(* CoDeSys 2.3.9.47 project: samur_8_8_16.pro *)
(* Libraries: STANDARD.LIB 5.6.98 12:03:02 *)

(* Task configuration *)
TASK Standard (PRIORITY := 0, INTERVAL := T#10ms);
	MAIN
END_TASK

(* Global variable list: TwinCAT_Configuration *)
(* Generated automatically by TwinCAT - (read only) *)
VAR_CONFIG
	CCB_FirstFloor.FCU_CCB1_23A_status AT %IX9.4 : BOOL;
	CCB_FirstFloor.FCU_CCB1_23A_trip AT %IX9.5 : BOOL;
	CCB_FirstFloor.FCU_CCB1_23A_mode AT %IX9.6 : BOOL;
	CCB_FirstFloor.FCU_CCB1_23A_FB.DEV1.AHU1_Relay AT %QX3.4 : BOOL;
	CCB_FirstFloor.FCU_CCB1_23B_status AT %IX9.7 : BOOL;
	CCB_FirstFloor.FCU_CCB1_23B_trip AT %IX10.0 : BOOL;
	CCB_FirstFloor.FCU_CCB1_23B_mode AT %IX10.1 : BOOL;
	CCB_FirstFloor.FCU_CCB1_23B_FB.DEV1.AHU1_Relay AT %QX3.5 : BOOL;
	CCB_FirstFloor.FCU_CCB1_23C_status AT %IX10.2 : BOOL;
	CCB_FirstFloor.FCU_CCB1_23C_trip AT %IX10.3 : BOOL;
	CCB_FirstFloor.FCU_CCB1_23C_mode AT %IX10.4 : BOOL;
	CCB_FirstFloor.FCU_CCB1_23C_FB.DEV1.AHU1_Relay AT %QX3.6 : BOOL;
	CCB_FirstFloor.DCS_Occupied AT %QX0.2 : BOOL;
	CCB_FirstFloor.common_alarm AT %QX0.3 : BOOL;
	CCB_GroundFloor.AHU_CCBG_01_status AT %IX0.0 : BOOL;
	CCB_GroundFloor.AHU_CCBG_01_trip AT %IX0.1 : BOOL;
	CCB_GroundFloor.AHU_CCBG_01_mode AT %IX0.2 : BOOL;
	CCB_GroundFloor.AHU_CCBG_01_belt AT %IX0.3 : BOOL;
	CCB_GroundFloor.AHU_CCBG_01_fire AT %IX0.4 : BOOL;
	CCB_GroundFloor.AHU_CCBG_01_gas AT %IX0.5 : BOOL;
	CCB_GroundFloor.AHU_CCBG_01_smoke AT %IX0.6 : BOOL;
	CCB_GroundFloor.AHU_CCBG_02_status AT %IX0.7 : BOOL;
	CCB_GroundFloor.AHU_CCBG_02_trip AT %IX1.0 : BOOL;
	CCB_GroundFloor.AHU_CCBG_02_mode AT %IX1.1 : BOOL;
	CCB_GroundFloor.AHU_CCBG_02_belt AT %IX1.2 : BOOL;
	CCB_GroundFloor.AHU_CCBG_02_fire AT %IX1.3 : BOOL;
	CCB_GroundFloor.AHU_CCBG_02_gas AT %IX1.4 : BOOL;
	CCB_GroundFloor.AHU_CCBG_02_smoke AT %IX1.5 : BOOL;
	CCB_GroundFloor.AHU_CCBG_03_status AT %IX1.6 : BOOL;
	CCB_GroundFloor.AHU_CCBG_03_trip AT %IX1.7 : BOOL;
	CCB_GroundFloor.AHU_CCBG_03_mode AT %IX2.0 : BOOL;
	CCB_GroundFloor.AHU_CCBG_03_belt AT %IX2.1 : BOOL;
	CCB_GroundFloor.AHU_CCBG_03_fire AT %IX2.2 : BOOL;
	CCB_GroundFloor.AHU_CCBG_03_gas AT %IX2.3 : BOOL;
	CCB_GroundFloor.AHU_CCBG_03_smoke AT %IX2.4 : BOOL;
	CCB_GroundFloor.AHU_CCCBG.DEV_1.AHU1_Relay AT %QX1.7 : BOOL;
	CCB_GroundFloor.AHU_CCCBG.DEV_2.AHU1_Relay AT %QX2.0 : BOOL;
	CCB_GroundFloor.AHU_CCCBG.DEV_3.AHU1_Relay AT %QX2.1 : BOOL;
	CCB_GroundFloor.EF_CCB_1_status AT %IX2.5 : BOOL;
	CCB_GroundFloor.EF_CCB_1_trip AT %IX2.6 : BOOL;
	CCB_GroundFloor.EF_CCB_1_mode AT %IX2.7 : BOOL;
	CCB_GroundFloor.EF_CCB_2_status AT %IX3.0 : BOOL;
	CCB_GroundFloor.EF_CCB_2_trip AT %IX3.1 : BOOL;
	CCB_GroundFloor.EF_CCB_2_mode AT %IX3.2 : BOOL;
	CCB_GroundFloor.EF_CCB.DEV_1.AHU1_Relay AT %QX2.2 : BOOL;
	CCB_GroundFloor.EF_CCB.DEV_2.AHU1_Relay AT %QX2.3 : BOOL;
	CCB_GroundFloor.TEF_CCB_01_status AT %IX3.3 : BOOL;
	CCB_GroundFloor.TEF_CCB_01_trip AT %IX3.4 : BOOL;
	CCB_GroundFloor.TEF_CCB_01_mode AT %IX3.5 : BOOL;
	CCB_GroundFloor.TEC_CCB.DEV1.AHU1_Relay AT %QX2.5 : BOOL;
	CCB_GroundFloor.EF_CCB_7A_status AT %IX3.6 : BOOL;
	CCB_GroundFloor.EF_CCB_7A_trip AT %IX3.7 : BOOL;
	CCB_GroundFloor.EF_CCB_7B_status AT %IX4.0 : BOOL;
	CCB_GroundFloor.EF_CCB_7B_trip AT %IX4.1 : BOOL;
	CCB_GroundFloor.EF_CCB_08_status AT %IX4.2 : BOOL;
	CCB_GroundFloor.EF_CCB_08_trip AT %IX4.3 : BOOL;
	CCB_GroundFloor.EH_CCB_01_flow_status AT %IX4.5 : BOOL;
	CCB_GroundFloor.EH_CCB_01_high_temp AT %IX4.6 : BOOL;
	CCB_GroundFloor.EH_CCB_01_FB.TEMPERATURE AT %IB32 : INT;
	CCB_GroundFloor.EH_CCB_01_FB.HEATER_STAGE1 AT %QX2.6 : BOOL;
	CCB_GroundFloor.EH_CCB_01_FB.HEATER_STAGE2 AT %QX2.7 : BOOL;
	CCB_GroundFloor.EH_CCB_01_FB.HEATER_STAGE3 AT %QX3.0 : BOOL;
	CCB_GroundFloor.EH_CCB_02_flow_status AT %IX5.0 : BOOL;
	CCB_GroundFloor.EH_CCB_02_high_temp AT %IX5.1 : BOOL;
	CCB_GroundFloor.EH_CCB_02_FB.TEMPERATURE AT %IB34 : INT;
	CCB_GroundFloor.EH_CCB_02_FB.HEATER_STAGE1 AT %QX3.1 : BOOL;
	CCB_GroundFloor.EH_CCB_02_FB.HEATER_STAGE2 AT %QX3.2 : BOOL;
	CCB_GroundFloor.EH_CCB_02_FB.HEATER_STAGE3 AT %QX3.3 : BOOL;
	CCB_GroundFloor.MD_CCBG_1_damper_open AT %IX5.2 : BOOL;
	CCB_GroundFloor.MD_CCBG_1_damper_close AT %IX5.3 : BOOL;
	CCB_GroundFloor.MD_CCBG_2_damper_open AT %IX5.4 : BOOL;
	CCB_GroundFloor.MD_CCBG_2_damper_close AT %IX5.5 : BOOL;
	CCB_GroundFloor.MD_CCBG_3_damper_open AT %IX5.6 : BOOL;
	CCB_GroundFloor.MD_CCBG_3_damper_close AT %IX5.7 : BOOL;
	CCB_GroundFloor.MD_CCBG_4_damper_open AT %IX6.0 : BOOL;
	CCB_GroundFloor.MD_CCBG_4_damper_close AT %IX6.1 : BOOL;
	CCB_GroundFloor.MD_EF_CCB_7A_damper_open AT %IX6.2 : BOOL;
	CCB_GroundFloor.MD_EF_CCB_7A_damper_close AT %IX6.3 : BOOL;
	CCB_GroundFloor.MD_EF_CCB_7B_damper_open AT %IX6.4 : BOOL;
	CCB_GroundFloor.MD_EF_CCB_7B_damper_close AT %IX6.5 : BOOL;
	CCB_GroundFloor.MD_EF_CCB_8_damper_open AT %IX6.6 : BOOL;
	CCB_GroundFloor.MD_EF_CCB_8_damper_close AT %IX6.7 : BOOL;
	CCB_GroundFloor.MFD_CCB_1_damper_open AT %IX7.0 : BOOL;
	CCB_GroundFloor.MFD_CCB_1_damper_close AT %IX7.1 : BOOL;
	CCB_GroundFloor.MFD_CCB_2_damper_open AT %IX7.2 : BOOL;
	CCB_GroundFloor.MFD_CCB_2_damper_close AT %IX7.3 : BOOL;
	CCB_GroundFloor.MFD_CCB_3_damper_open AT %IX7.4 : BOOL;
	CCB_GroundFloor.MFD_CCB_3_damper_close AT %IX7.5 : BOOL;
	CCB_GroundFloor.MFD_CCB_4_damper_open AT %IX7.6 : BOOL;
	CCB_GroundFloor.MFD_CCB_4_damper_close AT %IX7.7 : BOOL;
	CCB_GroundFloor.MFD_CCB_5_damper_open AT %IX8.0 : BOOL;
	CCB_GroundFloor.MFD_CCB_5_damper_close AT %IX8.1 : BOOL;
	CCB_GroundFloor.MFD_CCB_6_damper_open AT %IX8.2 : BOOL;
	CCB_GroundFloor.MFD_CCB_6_damper_close AT %IX8.3 : BOOL;
	CCB_GroundFloor.MFD_CCB_7_damper_open AT %IX8.4 : BOOL;
	CCB_GroundFloor.MFD_CCB_7_damper_close AT %IX8.5 : BOOL;
	CCB_GroundFloor.MFD_CCB_8_damper_open AT %IX8.6 : BOOL;
	CCB_GroundFloor.MFD_CCB_8_damper_close AT %IX8.7 : BOOL;
	CCB_GroundFloor.MFD_CCB_9_damper_open AT %IX9.0 : BOOL;
	CCB_GroundFloor.MFD_CCB_9_damper_close AT %IX9.1 : BOOL;
	CCB_GroundFloor.MFD_CCB_10_damper_open AT %IX9.2 : BOOL;
	CCB_GroundFloor.MFD_CCB_10_damper_close AT %IX9.3 : BOOL;
	CCB_GroundFloor.DCS_Occupied AT %QX0.0 : BOOL;
	CCB_GroundFloor.common_alarm AT %QX0.1 : BOOL;
	EDG_HOUSE.FB_AHU_EDG.DEV_1.AHU1_Relay AT %QX3.7 : BOOL;
	EDG_HOUSE.FB_AHU_EDG.DEV_2.AHU1_Relay AT %QX4.0 : BOOL;
	EDG_HOUSE.AHU_EDG_1_status AT %IX24.0 : BOOL;
	EDG_HOUSE.AHU_EDG_1_trip AT %IX24.1 : BOOL;
	EDG_HOUSE.AHU_EDG_1_mode AT %IX24.2 : BOOL;
	EDG_HOUSE.AHU_EDG_1_belt AT %IX24.3 : BOOL;
	EDG_HOUSE.AHU_EDG_1_fire AT %IX24.4 : BOOL;
	EDG_HOUSE.AHU_EDG_1_gas AT %IX24.5 : BOOL;
	EDG_HOUSE.AHU_EDG_1_smoke AT %IX24.6 : BOOL;
	EDG_HOUSE.AHU_EDG_2_status AT %IX24.7 : BOOL;
	EDG_HOUSE.AHU_EDG_2_trip AT %IX25.0 : BOOL;
	EDG_HOUSE.AHU_EDG_2_mode AT %IX25.1 : BOOL;
	EDG_HOUSE.AHU_EDG_2_belt AT %IX25.2 : BOOL;
	EDG_HOUSE.AHU_EDG_2_fire AT %IX25.3 : BOOL;
	EDG_HOUSE.AHU_EDG_2_gas AT %IX25.4 : BOOL;
	EDG_HOUSE.AHU_EDG_2_smoke AT %IX25.5 : BOOL;
	EDG_HOUSE.FB_EF_EDG.DEV_1.AHU1_Relay AT %QX4.2 : BOOL;
	EDG_HOUSE.FB_EF_EDG.DEV_2.AHU1_Relay AT %QX4.3 : BOOL;
	EDG_HOUSE.EF_EDG_1A_status AT %IX26.5 : BOOL;
	EDG_HOUSE.EF_EDG_1A_trip AT %IX26.6 : BOOL;
	EDG_HOUSE.EF_EDG_1A_mode AT %IX26.7 : BOOL;
	EDG_HOUSE.EF_EDG_1B_status AT %IX27.0 : BOOL;
	EDG_HOUSE.EF_EDG_1B_trip AT %IX27.1 : BOOL;
	EDG_HOUSE.EF_EDG_1B_mode AT %IX27.2 : BOOL;
	EDG_HOUSE.EF_EDG_2_status AT %IX27.3 : BOOL;
	EDG_HOUSE.EF_EDG_2_trip AT %IX27.4 : BOOL;
	EDG_HOUSE.EF_EDG_2_mode AT %IX27.5 : BOOL;
	EDG_HOUSE.MD_EDG_1A_damper_open AT %IX27.6 : BOOL;
	EDG_HOUSE.MD_EDG_1A_damper_close AT %IX27.7 : BOOL;
	EDG_HOUSE.MD_EDG_1B_damper_open AT %IX28.0 : BOOL;
	EDG_HOUSE.MD_EDG_1B_damper_close AT %IX28.1 : BOOL;
	EDG_HOUSE.MD_EF_EDG_2_damper_open AT %IX28.2 : BOOL;
	EDG_HOUSE.MD_EF_EDG_2_damper_close AT %IX28.3 : BOOL;
	EDG_HOUSE.MFD_EDG_1_damper_open AT %IX28.4 : BOOL;
	EDG_HOUSE.MFD_EDG_1_damper_close AT %IX28.5 : BOOL;
	EDG_HOUSE.MFD_EDG_2_damper_open AT %IX28.6 : BOOL;
	EDG_HOUSE.MFD_EDG_2_damper_close AT %IX28.7 : BOOL;
	EDG_HOUSE.MFD_EDG_3_damper_open AT %IX29.0 : BOOL;
	EDG_HOUSE.MFD_EDG_3_damper_close AT %IX29.1 : BOOL;
	Laboratory.AHU_LAB_1_status AT %IX10.5 : BOOL;
	Laboratory.AHU_LAB_1_trip AT %IX10.6 : BOOL;
	Laboratory.AHU_LAB_1_mode AT %IX10.7 : BOOL;
	Laboratory.AHU_LAB_1_belt AT %IX11.0 : BOOL;
	Laboratory.AHU_LAB_1_fire AT %IX11.1 : BOOL;
	Laboratory.AHU_LAB_1_gas AT %IX11.2 : BOOL;
	Laboratory.AHU_LAB_1_smoke AT %IX11.3 : BOOL;
	Laboratory.AHU_LAB_2_status AT %IX11.4 : BOOL;
	Laboratory.AHU_LAB_2_trip AT %IX11.5 : BOOL;
	Laboratory.AHU_LAB_2_mode AT %IX11.6 : BOOL;
	Laboratory.AHU_LAB_2_belt AT %IX11.7 : BOOL;
	Laboratory.AHU_LAB_2_fire AT %IX12.0 : BOOL;
	Laboratory.AHU_LAB_2_gas AT %IX12.1 : BOOL;
	Laboratory.AHU_LAB_2_smoke AT %IX12.2 : BOOL;
	Laboratory.AHU_LAB_3_status AT %IX12.3 : BOOL;
	Laboratory.AHU_LAB_3_trip AT %IX12.4 : BOOL;
	Laboratory.AHU_LAB_3_mode AT %IX12.5 : BOOL;
	Laboratory.AHU_LAB_3_belt AT %IX12.6 : BOOL;
	Laboratory.AHU_LAB_3_fire AT %IX12.7 : BOOL;
	Laboratory.AHU_LAB_3_gas AT %IX13.0 : BOOL;
	Laboratory.AHU_LAB_3_smoke AT %IX13.1 : BOOL;
	Laboratory.EF_LAB_1_status AT %IX13.2 : BOOL;
	Laboratory.EF_LAB_1_trip AT %IX13.3 : BOOL;
	Laboratory.EF_LAB_1_mode AT %IX13.4 : BOOL;
	Laboratory.EF_LAB_2_status AT %IX13.5 : BOOL;
	Laboratory.EF_LAB_2_trip AT %IX13.6 : BOOL;
	Laboratory.EF_LAB_2_mode AT %IX13.7 : BOOL;
	Laboratory.EF_LAB_3_status AT %IX14.0 : BOOL;
	Laboratory.EF_LAB_3_trip AT %IX14.1 : BOOL;
	Laboratory.EF_LAB_3_mode AT %IX14.2 : BOOL;
	Laboratory.EH_LAB_1_flow_status AT %IX14.4 : BOOL;
	Laboratory.EH_LAB_1_high_temp AT %IX14.5 : BOOL;
	Laboratory.MD_LAB_1_damper_open AT %IX14.6 : BOOL;
	Laboratory.MD_LAB_1_damper_close AT %IX14.7 : BOOL;
	Laboratory.MD_LAB_2_damper_open AT %IX15.0 : BOOL;
	Laboratory.MD_LAB_2_damper_close AT %IX15.1 : BOOL;
	Laboratory.MD_LAB_3_damper_open AT %IX15.2 : BOOL;
	Laboratory.MD_LAB_3_damper_close AT %IX15.3 : BOOL;
	Laboratory.MD_LAB_4_damper_open AT %IX15.4 : BOOL;
	Laboratory.MD_LAB_4_damper_close AT %IX15.5 : BOOL;
	TEST.fbTest_Flowchart_1_2.bAHU1_Status AT %IX29.2 : BOOL;
	TEST.fbTest_Flowchart_1_2.bAHU1_Trip AT %IX29.3 : BOOL;
	TEST.fbTest_Flowchart_1_2.bAHU1_Relay AT %QX0.4 : BOOL;
	TEST.fbTest_Flowchart_1_2.bAHU2_Status AT %IX29.4 : BOOL;
	TEST.fbTest_Flowchart_1_2.bAHU2_Trip AT %IX29.5 : BOOL;
	TEST.fbTest_Flowchart_1_2.bAHU2_Relay AT %QX0.5 : BOOL;
	TEST.fbTest_Flowchart_1_2.AHU1_DcsOccupied AT %QX0.6 : BOOL;
	TEST.fbTest_Flowchart_1_2.AHU1_StatusError AT %QX0.7 : BOOL;
	TEST.fbTest_Flowchart_1_2.AHU1_TripError AT %QX1.0 : BOOL;
	TEST.fbTest_Flowchart_1_2.AHU2_DcsOccupied AT %QX1.1 : BOOL;
	TEST.fbTest_Flowchart_1_2.AHU2_StatusError AT %QX1.2 : BOOL;
	TEST.fbTest_Flowchart_1_2.AHU2_TripError AT %QX1.3 : BOOL;
	TEST.fbtest.TEMPERATURE AT %IB30 : INT;
	TEST.fbtest.HEATER_STAGE1 AT %QX1.4 : BOOL;
	TEST.fbtest.HEATER_STAGE2 AT %QX1.5 : BOOL;
	TEST.fbtest.HEATER_STAGE3 AT %QX1.6 : BOOL;
END_VAR

(* POU MAIN, CFC *)
PROGRAM MAIN
VAR
END_VAR
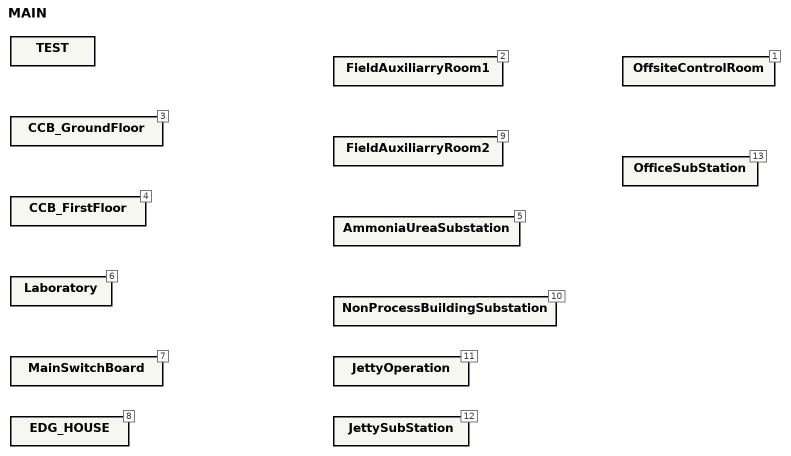
_CFC_ (* Continuous Function Chart, elements in execution order *)
#0 TEST()
#1 OffsiteControlRoom()
#2 FieldAuxiliarryRoom1()
#3 CCB_GroundFloor()
#4 CCB_FirstFloor()
#5 AmmoniaUreaSubstation()
#6 Laboratory()
#7 MainSwitchBoard()
#8 EDG_HOUSE()
#9 FieldAuxiliarryRoom2()
#10 NonProcessBuildingSubstation()
#11 JettyOperation()
#12 JettySubStation()
#13 OfficeSubStation()
_END_CFC_
(* the same logic as Structured Text *)
TEST();
OffsiteControlRoom();
FieldAuxiliarryRoom1();
CCB_GroundFloor();
CCB_FirstFloor();
AmmoniaUreaSubstation();
Laboratory();
MainSwitchBoard();
EDG_HOUSE();
FieldAuxiliarryRoom2();
NonProcessBuildingSubstation();
JettyOperation();
JettySubStation();
OfficeSubStation();
END_PROGRAM

(* POU GarbageCan/TEST, CFC *)
PROGRAM TEST
VAR
	fbTest_Flowchart_1_2: Flowchart_3_4_SingleButton;
	bAHU1: BOOL;
	bAHU2: BOOL;
	bAHU3: BOOL;

	fbtest: Flowchart_5_6;
END_VAR
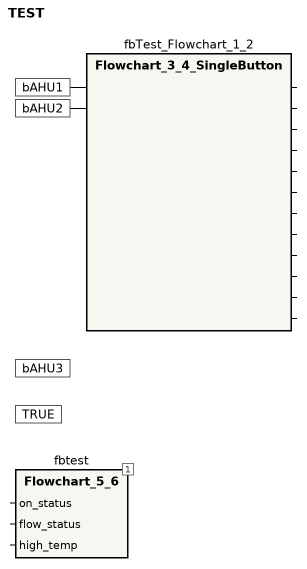
_CFC_ (* Continuous Function Chart, elements in execution order *)
#0 fbTest_Flowchart_1_2:Flowchart_3_4_SingleButton(bAHU1, bAHU2)
unconnected input bAHU3
unconnected input TRUE
#1 fbtest:Flowchart_5_6(on_status: -, flow_status: -, high_temp: -)
_END_CFC_
(* the same logic as Structured Text *)
fbTest_Flowchart_1_2(bAHU1, bAHU2);
fbtest();
END_PROGRAM

(* POU GarbageCan/Flowchart_3_4_SingleButton, CFC *)
FUNCTION_BLOCK Flowchart_3_4_SingleButton
VAR_INPUT
END_VAR
VAR_OUTPUT
	AHU1_DcsOccupied AT%Q*: BOOL;
	AHU1_StatusError  AT%Q*: BOOL;
	AHU1_TripError AT%Q*: BOOL;
	bAHU1_Error: BOOL;

	AHU2_DcsOccupied AT%Q*: BOOL;
	AHU2_StatusError  AT%Q*: BOOL;
	AHU2_TripError AT%Q*: BOOL;
	bAHU2_Error: BOOL;

	AHU_CommonAlarm:BOOL;
	AHU_DCSOccupied:BOOL;

END_VAR
VAR




	bAHU1_Status AT %I*: BOOL;
	bAHU1_Trip AT %I*: BOOL;
	bAHU1_Relay AT %Q*: BOOL;
	Status_timer_1: TON;
	Error_timer_1: TOF;
	OnRtrigAHU1: R_TRIG;
	OffRtrigAHU1: R_TRIG;


	bAHU2_Status AT %I*: BOOL;
	bAHU2_Trip AT %I*: BOOL;
	bAHU2_Relay AT %Q*: BOOL;
	Status_timer_2: TON;
	Error_timer_2: TOF;
	OnRtrigAHU2: R_TRIG;
	OffRtrigAHU2: R_TRIG;


	AHU1_Reset: TON;
	AHU2_Reset: TON;
END_VAR
VAR_IN_OUT
	bAHU1_On: BOOL;
	bAHU2_On: BOOL;

END_VAR
VAR (* helpers for the ST form of the networks *)
	_t14 : BOOL;
	_t65 : BOOL;
	_t137 : BOOL;
	_t152 : BOOL;
END_VAR
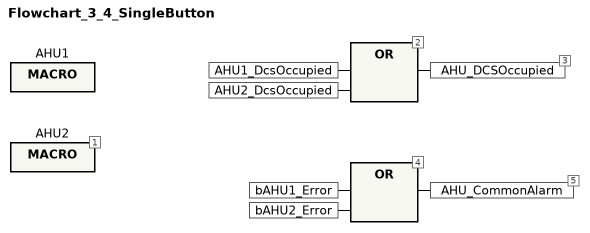
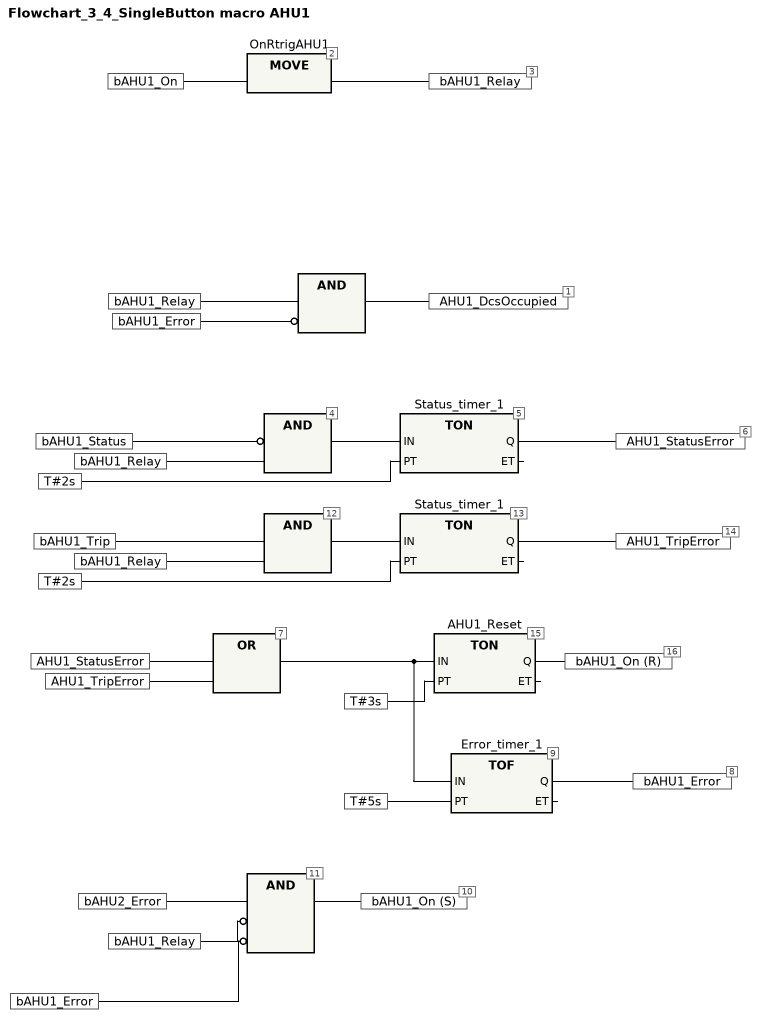
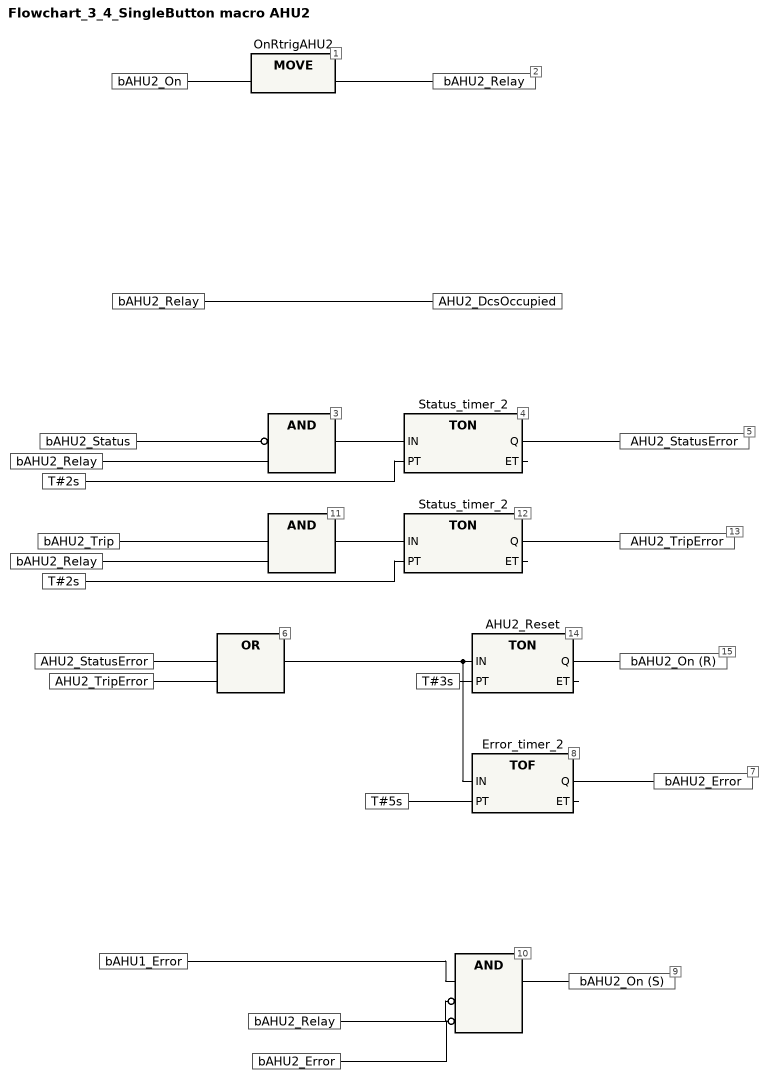
_CFC_ (* Continuous Function Chart, elements in execution order *)
#0 MACRO AHU1()
	#1 AND(bAHU1_Relay, NOT bAHU1_Error)
	#2 AHU1_DcsOccupied <= #1
	#3 OnRtrigAHU1:MOVE(bAHU1_On)
	#4 bAHU1_Relay <= #3
	#5 AND(NOT bAHU1_Status, bAHU1_Relay)
	#6 Status_timer_1:TON(IN: #5, PT: T#2s)
	#7 AHU1_StatusError <= #6.Q
	#8 OR(AHU1_StatusError, AHU1_TripError)
	#9 bAHU1_Error <= #10.Q
	#10 Error_timer_1:TOF(IN: #8, PT: T#5s)
	#11 S bAHU1_On <= #12
	#12 AND(bAHU2_Error, NOT bAHU1_Relay, NOT bAHU1_Error)
	#13 AND(bAHU1_Trip, bAHU1_Relay)
	#14 Status_timer_1:TON(IN: #13, PT: T#2s)
	#15 AHU1_TripError <= #14.Q
	#16 AHU1_Reset:TON(IN: #8, PT: T#3s)
	#17 R bAHU1_On <= #16.Q
END_MACRO
#18 MACRO AHU2()
	#19 AHU2_DcsOccupied <= bAHU2_Relay
	#20 OnRtrigAHU2:MOVE(bAHU2_On)
	#21 bAHU2_Relay <= #20
	#22 AND(NOT bAHU2_Status, bAHU2_Relay)
	#23 Status_timer_2:TON(IN: #22, PT: T#2s)
	#24 AHU2_StatusError <= #23.Q
	#25 OR(AHU2_StatusError, AHU2_TripError)
	#26 bAHU2_Error <= #27.Q
	#27 Error_timer_2:TOF(IN: #25, PT: T#5s)
	#28 S bAHU2_On <= #29
	#29 AND(bAHU1_Error, NOT bAHU2_Relay, NOT bAHU2_Error)
	#30 AND(bAHU2_Trip, bAHU2_Relay)
	#31 Status_timer_2:TON(IN: #30, PT: T#2s)
	#32 AHU2_TripError <= #31.Q
	#33 AHU2_Reset:TON(IN: #25, PT: T#3s)
	#34 R bAHU2_On <= #33.Q
END_MACRO
#35 OR(AHU1_DcsOccupied, AHU2_DcsOccupied)
#36 AHU_DCSOccupied <= #35
#37 OR(bAHU1_Error, bAHU2_Error)
#38 AHU_CommonAlarm <= #37
_END_CFC_
(* the same logic as Structured Text *)
(* macro AHU1 *)
AHU1_DcsOccupied := bAHU1_Relay AND NOT bAHU1_Error;
bAHU1_Relay := bAHU1_On;
Status_timer_1(IN := NOT bAHU1_Status AND bAHU1_Relay, PT := T#2s);
AHU1_StatusError := Status_timer_1.Q;
_t14 := AHU1_StatusError OR AHU1_TripError;
bAHU1_Error := Error_timer_1.Q;
Error_timer_1(IN := _t14, PT := T#5s);
IF _t65 THEN bAHU1_On := TRUE; END_IF;
_t65 := bAHU2_Error AND NOT bAHU1_Relay AND NOT bAHU1_Error;
Status_timer_1(IN := bAHU1_Trip AND bAHU1_Relay, PT := T#2s);
AHU1_TripError := Status_timer_1.Q;
AHU1_Reset(IN := _t14, PT := T#3s);
IF AHU1_Reset.Q THEN bAHU1_On := FALSE; END_IF;
(* macro AHU2 *)
AHU2_DcsOccupied := bAHU2_Relay;
bAHU2_Relay := bAHU2_On;
Status_timer_2(IN := NOT bAHU2_Status AND bAHU2_Relay, PT := T#2s);
AHU2_StatusError := Status_timer_2.Q;
_t137 := AHU2_StatusError OR AHU2_TripError;
bAHU2_Error := Error_timer_2.Q;
Error_timer_2(IN := _t137, PT := T#5s);
IF _t152 THEN bAHU2_On := TRUE; END_IF;
_t152 := bAHU1_Error AND NOT bAHU2_Relay AND NOT bAHU2_Error;
Status_timer_2(IN := bAHU2_Trip AND bAHU2_Relay, PT := T#2s);
AHU2_TripError := Status_timer_2.Q;
AHU2_Reset(IN := _t137, PT := T#3s);
IF AHU2_Reset.Q THEN bAHU2_On := FALSE; END_IF;
AHU_DCSOccupied := AHU1_DcsOccupied OR AHU2_DcsOccupied;
AHU_CommonAlarm := bAHU1_Error OR bAHU2_Error;
END_FUNCTION_BLOCK

(* POU Module/Flowchart_5_6, CFC *)
FUNCTION_BLOCK Flowchart_5_6
VAR_INPUT
	on_status 			:BOOL;
	flow_status			: BOOL;
	high_temp 			: BOOL;
END_VAR
VAR_OUTPUT
END_VAR
VAR
	TEMPERATURE		AT%I*: INT;
	HEATER_STAGE1	AT%Q* : BOOL;
	HEATER_STAGE2 	AT%Q*: BOOL;
	HEATER_STAGE3 	AT%Q*: BOOL;
END_VAR
VAR (* helpers for the ST form of the networks *)
	_t2 : BOOL;
END_VAR
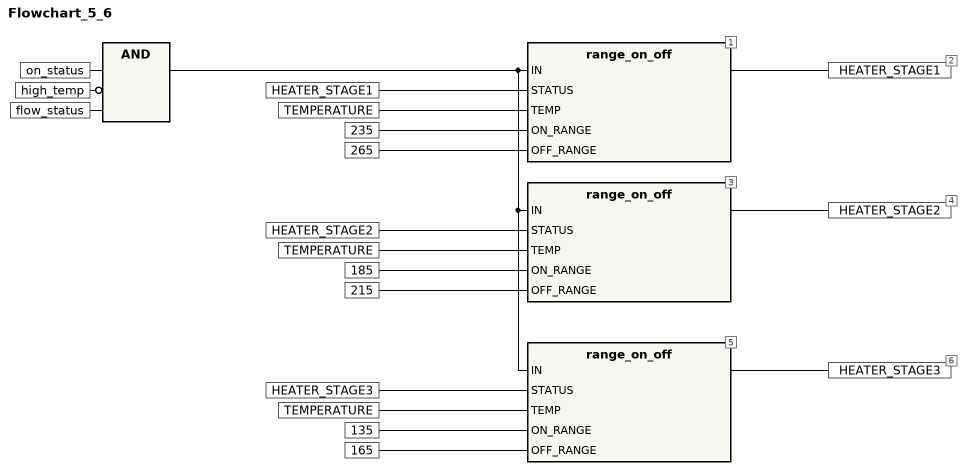
_CFC_ (* Continuous Function Chart, elements in execution order *)
#0 AND(on_status, NOT high_temp, flow_status)
#1 range_on_off(IN: #0, STATUS: HEATER_STAGE1, TEMP: TEMPERATURE, ON_RANGE: 235, OFF_RANGE: 265)
#2 HEATER_STAGE1 <= #1
#3 range_on_off(IN: #0, STATUS: HEATER_STAGE2, TEMP: TEMPERATURE, ON_RANGE: 185, OFF_RANGE: 215)
#4 HEATER_STAGE2 <= #3
#5 range_on_off(IN: #0, STATUS: HEATER_STAGE3, TEMP: TEMPERATURE, ON_RANGE: 135, OFF_RANGE: 165)
#6 HEATER_STAGE3 <= #5
_END_CFC_
(* the same logic as Structured Text *)
_t2 := on_status AND NOT high_temp AND flow_status;
HEATER_STAGE1 := range_on_off(IN := _t2, STATUS := HEATER_STAGE1, TEMP := TEMPERATURE, ON_RANGE := 235, OFF_RANGE := 265);
HEATER_STAGE2 := range_on_off(IN := _t2, STATUS := HEATER_STAGE2, TEMP := TEMPERATURE, ON_RANGE := 185, OFF_RANGE := 215);
HEATER_STAGE3 := range_on_off(IN := _t2, STATUS := HEATER_STAGE3, TEMP := TEMPERATURE, ON_RANGE := 135, OFF_RANGE := 165);
END_FUNCTION_BLOCK

(* POU Module/range_on_off, ST *)
FUNCTION range_on_off : BOOL
VAR_INPUT
	IN : BOOL;
	STATUS : BOOL;
	TEMP : INT;
	ON_RANGE : INT;
	OFF_RANGE : INT;

END_VAR
VAR
END_VAR
IF STATUS THEN
	IF TEMP >= OFF_RANGE THEN
		range_on_off := FALSE;
	ELSE
		range_on_off := IN;
	END_IF
ELSE
	IF TEMP < ON_RANGE THEN
		range_on_off := IN;
	ELSE
		range_on_off := FALSE;
	END_IF
END_IF
END_FUNCTION

(* POU OffsiteControlRoom, ST *)
PROGRAM OffsiteControlRoom
VAR
	AHU_OFFCR_common_alarm : BOOL;
	AHU_OFFCR_dcs_occupied : BOOL;

	AHU_OFFCR_dummy : BOOL;
	FB_AHU_OFFCR: Flowchart_3_4_CTRL;

	AHU_OFFCR_1_status AT%I* : BOOL;
	AHU_OFFCR_1_trip AT%I* : BOOL;
	AHU_OFFCR_1_mode AT%I* : BOOL;
	AHU_OFFCR_1_belt AT%I* : BOOL;
	AHU_OFFCR_1_fire AT%I* : BOOL;
	AHU_OFFCR_1_gas AT%I* : BOOL;
	AHU_OFFCR_1_smoke AT%I* : BOOL;

	AHU_OFFCR_1_trigger : BOOL;
	AHU_OFFCR_1_latch : BOOL;
	AHU_OFFCR_1_common_alarm : BOOL;
	AHU_OFFCR_1_status_error : BOOL;
	AHU_OFFCR_1_trip_error : BOOL;
	AHU_OFFCR_1_dcs_occupied : BOOL;

	AHU_OFFCR_1_status_Filter : ErrorFilter;
	AHU_OFFCR_1_trip_Filter : ErrorFilter;


	AHU_OFFCR_2_status AT%I* : BOOL;
	AHU_OFFCR_2_trip AT%I* : BOOL;
	AHU_OFFCR_2_mode AT%I* : BOOL;
	AHU_OFFCR_2_belt AT%I* : BOOL;
	AHU_OFFCR_2_fire AT%I* : BOOL;
	AHU_OFFCR_2_gas AT%I* : BOOL;
	AHU_OFFCR_2_smoke AT%I* : BOOL;

	AHU_OFFCR_2_trigger : BOOL;
	AHU_OFFCR_2_latch : BOOL;
	AHU_OFFCR_2_common_alarm : BOOL;
	AHU_OFFCR_2_status_error : BOOL;
	AHU_OFFCR_2_trip_error : BOOL;
	AHU_OFFCR_2_dcs_occupied : BOOL;

	AHU_OFFCR_2_status_Filter : ErrorFilter;
	AHU_OFFCR_2_trip_Filter : ErrorFilter;

(**************************************************)

	EF_OFFCR_common_alarm : BOOL;
	EF_OFFCR_dcs_occupied : BOOL;

	EF_OFFCR_dummy : BOOL;
	FB_EF_OFFCR: Flowchart_3_4_CTRL;

	EF_OFFCR_1A_status AT%I* : BOOL;
	EF_OFFCR_1A_trip AT%I* : BOOL;
	EF_OFFCR_1A_mode AT%I* : BOOL;

	EF_OFFCR_1A_trigger : BOOL;
	EF_OFFCR_1A_latch : BOOL;
	EF_OFFCR_1A_common_alarm : BOOL;
	EF_OFFCR_1A_status_error : BOOL;
	EF_OFFCR_1A_trip_error : BOOL;
	EF_OFFCR_1A_dcs_occupied : BOOL;

	EF_OFFCR_1A_status_Filter : ErrorFilter;
	EF_OFFCR_1A_trip_Filter : ErrorFilter;


	EF_OFFCR_1B_status AT%I* : BOOL;
	EF_OFFCR_1B_trip AT%I* : BOOL;
	EF_OFFCR_1B_mode AT%I* : BOOL;

	EF_OFFCR_1B_trigger : BOOL;
	EF_OFFCR_1B_latch : BOOL;
	EF_OFFCR_1B_common_alarm : BOOL;
	EF_OFFCR_1B_status_error : BOOL;
	EF_OFFCR_1B_trip_error : BOOL;
	EF_OFFCR_1B_dcs_occupied : BOOL;

	EF_OFFCR_1B_status_Filter : ErrorFilter;
	EF_OFFCR_1B_trip_Filter : ErrorFilter;

(*************************************************************)

	EF_OFFCR_common_alarm_2 : BOOL;
	EF_OFFCR_dcs_occupied_2 : BOOL;


	FB_EF_OFFCR_2: Flowchart_7;

	EF_OFFCR_2_status AT%I* : BOOL;
	EF_OFFCR_2_trip AT%I* : BOOL;
	EF_OFFCR_2_mode AT%I* : BOOL;

	EF_OFFCR_2_trigger : BOOL;
	EF_OFFCR_2_latch : BOOL;
	EF_OFFCR_2_common_alarm : BOOL;
	EF_OFFCR_2_status_error : BOOL;
	EF_OFFCR_2_trip_error : BOOL;
	EF_OFFCR_2_dcs_occupied : BOOL;

	EF_OFFCR_2_status_Filter : ErrorFilter;
	EF_OFFCR_2_trip_Filter : ErrorFilter;


	FB_EF_OFFCR_3: Flowchart_7;

	EF_OFFCR_3_status AT%I* : BOOL;
	EF_OFFCR_3_trip AT%I* : BOOL;
	EF_OFFCR_3_mode AT%I* : BOOL;

	EF_OFFCR_3_trigger : BOOL;
	EF_OFFCR_3_latch : BOOL;
	EF_OFFCR_3_common_alarm : BOOL;
	EF_OFFCR_3_status_error : BOOL;
	EF_OFFCR_3_trip_error : BOOL;
	EF_OFFCR_3_dcs_occupied : BOOL;

	EF_OFFCR_3_status_Filter : ErrorFilter;
	EF_OFFCR_3_trip_Filter : ErrorFilter;

(************************************************************)

	EF_OFFCR_common_alarm_3 : BOOL;


	EF_OFFCR_3A_status AT%I* : BOOL;
	EF_OFFCR_3A_trip AT%I* : BOOL;
	EF_OFFCR_3A_mode AT%I* : BOOL;

	EF_OFFCR_3A_trigger : BOOL;
	EF_OFFCR_3A_latch : BOOL;
	EF_OFFCR_3A_common_alarm : BOOL;
	EF_OFFCR_3A_status_error : BOOL;
	EF_OFFCR_3A_trip_error : BOOL;
	EF_OFFCR_3A_dcs_occupied : BOOL;

	EF_OFFCR_3A_status_Filter : ErrorFilter;
	EF_OFFCR_3A_trip_Filter : ErrorFilter;



	EF_OFFCR_3B_status AT%I* : BOOL;
	EF_OFFCR_3B_trip AT%I* : BOOL;
	EF_OFFCR_3B_mode AT%I* : BOOL;

	EF_OFFCR_3B_trigger : BOOL;
	EF_OFFCR_3B_latch : BOOL;
	EF_OFFCR_3B_common_alarm : BOOL;
	EF_OFFCR_3B_status_error : BOOL;
	EF_OFFCR_3B_trip_error : BOOL;
	EF_OFFCR_3B_dcs_occupied : BOOL;

	EF_OFFCR_3B_status_Filter : ErrorFilter;
	EF_OFFCR_3B_trip_Filter : ErrorFilter;




	EF_OFFCR_4A_status AT%I* : BOOL;
	EF_OFFCR_4A_trip AT%I* : BOOL;
	EF_OFFCR_4A_mode AT%I* : BOOL;

	EF_OFFCR_4A_trigger : BOOL;
	EF_OFFCR_4A_latch : BOOL;
	EF_OFFCR_4A_common_alarm : BOOL;
	EF_OFFCR_4A_status_error : BOOL;
	EF_OFFCR_4A_trip_error : BOOL;
	EF_OFFCR_4A_dcs_occupied : BOOL;

	EF_OFFCR_4A_status_Filter : ErrorFilter;
	EF_OFFCR_4A_trip_Filter : ErrorFilter;



	EF_OFFCR_4B_status AT%I* : BOOL;
	EF_OFFCR_4B_trip AT%I* : BOOL;
	EF_OFFCR_4B_mode AT%I* : BOOL;

	EF_OFFCR_4B_trigger : BOOL;
	EF_OFFCR_4B_latch : BOOL;
	EF_OFFCR_4B_common_alarm : BOOL;
	EF_OFFCR_4B_status_error : BOOL;
	EF_OFFCR_4B_trip_error : BOOL;
	EF_OFFCR_4B_dcs_occupied : BOOL;

	EF_OFFCR_4B_status_Filter : ErrorFilter;
	EF_OFFCR_4B_trip_Filter : ErrorFilter;


(********************************************************************)


	FB_EDH_OFFCR_1: Flowchart_5_6;
	EDH_OFFCR_1_on_status : BOOL;
	EDH_OFFCR_1_flow_status AT%I* : BOOL;
	EDH_OFFCR_1_high_temp AT%I* : BOOL;

	EDH_OFFCR_1_common_alarm : BOOL;
	EDH_OFFCR_1_hightemp_error : BOOL;

(*********************************************************)

	MD_OFFCR_1A_damper_open AT%I* : BOOL;
	MD_OFFCR_1A_damper_close AT%I* : BOOL;

	MD_OFFCR_1B_damper_open AT%I* : BOOL;
	MD_OFFCR_1B_damper_close AT%I* : BOOL;

	MD_OFFCR_1C_damper_open AT%I* : BOOL;
	MD_OFFCR_1C_damper_close AT%I* : BOOL;

	MD_OFFCR_2A_damper_open AT%I* : BOOL;
	MD_OFFCR_2A_damper_close AT%I* : BOOL;

	MD_OFFCR_2B_damper_open AT%I* : BOOL;
	MD_OFFCR_2B_damper_close AT%I* : BOOL;

	MD_OFFCR_3A_damper_open AT%I* : BOOL;
	MD_OFFCR_3A_damper_close AT%I* : BOOL;

	MD_OFFCR_3B_damper_open AT%I* : BOOL;
	MD_OFFCR_3B_damper_close AT%I* : BOOL;

(***********************************************************)


	MFD_OFFCR_1_damper_open AT%I* : BOOL;
	MFD_OFFCR_1_damper_close AT%I* : BOOL;

	MFD_OFFCR_2_damper_open AT%I* : BOOL;
	MFD_OFFCR_2_damper_close AT%I* : BOOL;

	MFD_OFFCR_3_damper_open AT%I* : BOOL;
	MFD_OFFCR_3_damper_close AT%I* : BOOL;

	MFD_OFFCR_4_damper_open AT%I* : BOOL;
	MFD_OFFCR_4_damper_close AT%I* : BOOL;

	MFD_OFFCR_5_damper_open AT%I* : BOOL;
	MFD_OFFCR_5_damper_close AT%I* : BOOL;

	MFD_OFFCR_6_damper_open AT%I* : BOOL;
	MFD_OFFCR_6_damper_close AT%I* : BOOL;

	MFD_OFFCR_7_damper_open AT%I* : BOOL;
	MFD_OFFCR_7_damper_close AT%I* : BOOL;

(********************************************************************)

	common_alarm AT%Q* : BOOL;
	dcs_occupied AT%Q* : BOOL;

END_VAR
AHU_OFFCR_1_status_Filter(IN:=(NOT AHU_OFFCR_1_status AND AHU_OFFCR_1_latch),Q=>AHU_OFFCR_1_status_error);
AHU_OFFCR_1_trip_Filter(IN:=(AHU_OFFCR_1_trip AND AHU_OFFCR_1_latch),Q=>AHU_OFFCR_1_trip_error);
AHU_OFFCR_1_common_alarm := AHU_OFFCR_1_fire OR AHU_OFFCR_1_gas OR AHU_OFFCR_1_smoke OR AHU_OFFCR_1_status_error OR AHU_OFFCR_1_trip_error;



AHU_OFFCR_2_status_Filter(IN:=(NOT AHU_OFFCR_2_status AND AHU_OFFCR_2_latch),Q=>AHU_OFFCR_2_status_error);
AHU_OFFCR_2_trip_Filter(IN:=(AHU_OFFCR_2_trip AND AHU_OFFCR_2_latch),Q=>AHU_OFFCR_2_trip_error);
AHU_OFFCR_2_common_alarm := AHU_OFFCR_2_fire OR AHU_OFFCR_2_gas OR AHU_OFFCR_2_smoke OR AHU_OFFCR_2_status_error OR AHU_OFFCR_2_trip_error;


AHU_OFFCR_common_alarm := AHU_OFFCR_1_common_alarm OR AHU_OFFCR_2_common_alarm;
AHU_OFFCR_dcs_occupied := AHU_OFFCR_1_dcs_occupied OR AHU_OFFCR_2_dcs_occupied;

	FB_AHU_OFFCR(
	ON1:=AHU_OFFCR_1_trigger ,
	ON2:=AHU_OFFCR_2_trigger ,
	ON3:=FALSE ,
	status_error_1:= AHU_OFFCR_1_status_error,
	status_error_2:=AHU_OFFCR_2_status_error ,
	status_error_3:=FALSE ,
	trip_error_1:=AHU_OFFCR_1_trip_error ,
	trip_error_2:=AHU_OFFCR_2_trip_error ,
	trip_error_3:=FALSE ,
	Latch1:=AHU_OFFCR_1_latch ,
	Latch2:=AHU_OFFCR_2_latch ,
	Latch3:=AHU_OFFCR_dummy ,
	DcsOccupied_1=>AHU_OFFCR_1_dcs_occupied ,
	DcsOccupied_2=>AHU_OFFCR_2_dcs_occupied ,
	DcsOccupied_3=> );

(*************************************************************)


EF_OFFCR_1A_status_Filter(IN:=(NOT EF_OFFCR_1A_status AND EF_OFFCR_1A_latch),Q=>EF_OFFCR_1A_status_error);
EF_OFFCR_1A_trip_Filter(IN:=(EF_OFFCR_1A_trip AND EF_OFFCR_1A_latch),Q=>EF_OFFCR_1A_trip_error);
EF_OFFCR_1A_common_alarm := EF_OFFCR_1A_status_error OR EF_OFFCR_1A_trip_error;

EF_OFFCR_1B_status_Filter(IN:=(NOT EF_OFFCR_1B_status AND EF_OFFCR_1B_latch),Q=>EF_OFFCR_1B_status_error);
EF_OFFCR_1B_trip_Filter(IN:=(EF_OFFCR_1B_trip AND EF_OFFCR_1B_latch),Q=>EF_OFFCR_1B_trip_error);
EF_OFFCR_1B_common_alarm := EF_OFFCR_1B_status_error OR EF_OFFCR_1B_trip_error;


EF_OFFCR_common_alarm := EF_OFFCR_1A_common_alarm OR EF_OFFCR_1B_common_alarm;
EF_OFFCR_dcs_occupied := EF_OFFCR_1A_dcs_occupied OR EF_OFFCR_1B_dcs_occupied;

	FB_EF_OFFCR(
	ON1:=EF_OFFCR_1A_trigger ,
	ON2:=EF_OFFCR_1B_trigger ,
	ON3:=FALSE ,
	status_error_1:= EF_OFFCR_1A_status_error,
	status_error_2:=EF_OFFCR_1B_status_error ,
	status_error_3:=FALSE ,
	trip_error_1:=EF_OFFCR_1A_trip_error ,
	trip_error_2:=EF_OFFCR_1B_trip_error ,
	trip_error_3:=FALSE ,
	Latch1:=EF_OFFCR_1A_latch ,
	Latch2:=EF_OFFCR_1B_latch ,
	Latch3:=EF_OFFCR_dummy ,
	DcsOccupied_1=>EF_OFFCR_1A_dcs_occupied ,
	DcsOccupied_2=>EF_OFFCR_1B_dcs_occupied ,
	DcsOccupied_3=> );

(***********************************************************)



EF_OFFCR_2_status_Filter(IN:=(NOT EF_OFFCR_2_status AND EF_OFFCR_2_latch),Q=>EF_OFFCR_2_status_error);
EF_OFFCR_2_trip_Filter(IN:=(EF_OFFCR_2_trip AND EF_OFFCR_2_latch),Q=>EF_OFFCR_2_trip_error);
EF_OFFCR_2_common_alarm := EF_OFFCR_2_status_error OR EF_OFFCR_2_trip_error;


FB_EF_OFFCR_2(
Trigger:=EF_OFFCR_2_trigger ,
Latch:=EF_OFFCR_2_latch ,
DCS_Occupied=>EF_OFFCR_2_dcs_occupied );



EF_OFFCR_common_alarm_2:=EF_OFFCR_2_common_alarm OR EF_OFFCR_3_common_alarm;
EF_OFFCR_dcs_occupied_2:=EF_OFFCR_2_dcs_occupied OR EF_OFFCR_3_dcs_occupied;

(************************************************************)

EF_OFFCR_3A_status_Filter(IN:=(NOT EF_OFFCR_3A_status AND EF_OFFCR_3A_latch),Q=>EF_OFFCR_3A_status_error);
EF_OFFCR_3A_trip_Filter(IN:=(EF_OFFCR_3A_trip AND EF_OFFCR_3A_latch),Q=>EF_OFFCR_3A_trip_error);
EF_OFFCR_3A_common_alarm := EF_OFFCR_3A_status_error OR EF_OFFCR_3A_trip_error;

EF_OFFCR_3B_status_Filter(IN:=(NOT EF_OFFCR_3B_status AND EF_OFFCR_3B_latch),Q=>EF_OFFCR_3B_status_error);
EF_OFFCR_3B_trip_Filter(IN:=(EF_OFFCR_3B_trip AND EF_OFFCR_3B_latch),Q=>EF_OFFCR_3B_trip_error);
EF_OFFCR_3B_common_alarm := EF_OFFCR_3B_status_error OR EF_OFFCR_3B_trip_error;

EF_OFFCR_4A_status_Filter(IN:=(NOT EF_OFFCR_4A_status AND EF_OFFCR_4A_latch),Q=>EF_OFFCR_4A_status_error);
EF_OFFCR_4A_trip_Filter(IN:=(EF_OFFCR_4A_trip AND EF_OFFCR_4A_latch),Q=>EF_OFFCR_4A_trip_error);
EF_OFFCR_4A_common_alarm := EF_OFFCR_4A_status_error OR EF_OFFCR_4A_trip_error;

EF_OFFCR_4B_status_Filter(IN:=(NOT EF_OFFCR_4B_status AND EF_OFFCR_4B_latch),Q=>EF_OFFCR_4B_status_error);
EF_OFFCR_4B_trip_Filter(IN:=(EF_OFFCR_4B_trip AND EF_OFFCR_4B_latch),Q=>EF_OFFCR_4B_trip_error);
EF_OFFCR_4B_common_alarm := EF_OFFCR_4B_status_error OR EF_OFFCR_4B_trip_error;



EF_OFFCR_common_alarm_3:=EF_OFFCR_4A_common_alarm OR EF_OFFCR_4B_common_alarm OR EF_OFFCR_3A_common_alarm OR EF_OFFCR_3B_common_alarm;

(****************************************************************************************)

EDH_OFFCR_1_on_status := AHU_OFFCR_dcs_occupied;
EDH_OFFCR_1_hightemp_error := EDH_OFFCR_1_high_temp;
EDH_OFFCR_1_common_alarm := EDH_OFFCR_1_hightemp_error;

FB_EDH_OFFCR_1(on_status:= EDH_OFFCR_1_on_status , flow_status:= EDH_OFFCR_1_flow_status , high_temp:= EDH_OFFCR_1_high_temp);

(****************************************************************************************)

common_alarm := AHU_OFFCR_common_alarm OR EF_OFFCR_common_alarm OR EF_OFFCR_common_alarm_2 OR EF_OFFCR_common_alarm_3 OR EDH_OFFCR_1_common_alarm;
dcs_occupied := AHU_OFFCR_dcs_occupied OR EF_OFFCR_dcs_occupied OR EF_OFFCR_dcs_occupied_2;
END_PROGRAM

(* POU Module/Flowchart_3_4_CTRL, CFC *)
FUNCTION_BLOCK Flowchart_3_4_CTRL
VAR
	DEV_1: AHU_INTERNAL;
	DEV_2: AHU_INTERNAL;

	DEV1_ErrorInternal_1: ERROR_INTERNAL;
	DEV1_ErrorInternal_2: ERROR_INTERNAL;

	DEV2_ErrorInternal_1: ERROR_INTERNAL;
	DEV2_ErrorInternal_2: ERROR_INTERNAL;

END_VAR
VAR_INPUT
	ON1: BOOL;
	ON2: BOOL;
	ON3: BOOL;

	status_error_1 : BOOL;
	status_error_2 : BOOL;
	status_error_3 : BOOL;

	trip_error_1 : BOOL;
	trip_error_2 : BOOL;
	trip_error_3 : BOOL;


END_VAR
VAR_IN_OUT
	Latch1:BOOL;
	Latch2:BOOL;
	Latch3:BOOL;
END_VAR
VAR_OUTPUT
	DcsOccupied_1: BOOL;
	DcsOccupied_2: BOOL;
	DcsOccupied_3: BOOL;
END_VAR
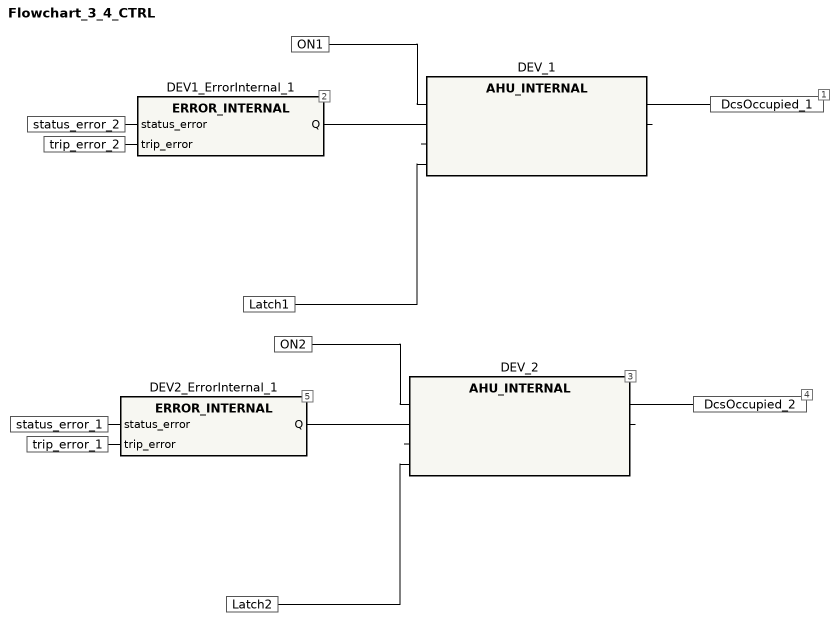
_CFC_ (* Continuous Function Chart, elements in execution order *)
#0 DEV_1:AHU_INTERNAL(ON1, #2.Q, -, Latch1)
#1 DcsOccupied_1 <= #0.out 1
#2 DEV1_ErrorInternal_1:ERROR_INTERNAL(status_error: status_error_2, trip_error: trip_error_2)
#3 DEV_2:AHU_INTERNAL(ON2, #5.Q, -, Latch2)
#4 DcsOccupied_2 <= #3.out 1
#5 DEV2_ErrorInternal_1:ERROR_INTERNAL(status_error: status_error_1, trip_error: trip_error_1)
_END_CFC_
END_FUNCTION_BLOCK

(* POU Module/AHU_INTERNAL, CFC *)
FUNCTION_BLOCK AHU_INTERNAL
VAR_INPUT
	AHU1_On: BOOL;
	Emergency1 : BOOL;
	Emergency2 : BOOL;
END_VAR
VAR_OUTPUT
	DcsOccupied : BOOL;
END_VAR
VAR
	AHU1_Relay AT %Q*: BOOL;

	Error_timer_1: TOF;
	OnRtrigAHU1: R_TRIG;
	OffRtrigAHU1: R_TRIG;
	Emergencylatch1: R_TRIG;
	Emergencylatch2: R_TRIG;
END_VAR
VAR_IN_OUT
	AHU1_Latch : BOOL;
END_VAR
VAR (* helpers for the ST form of the networks *)
	_t232 : BOOL;
END_VAR
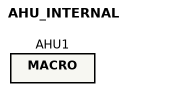
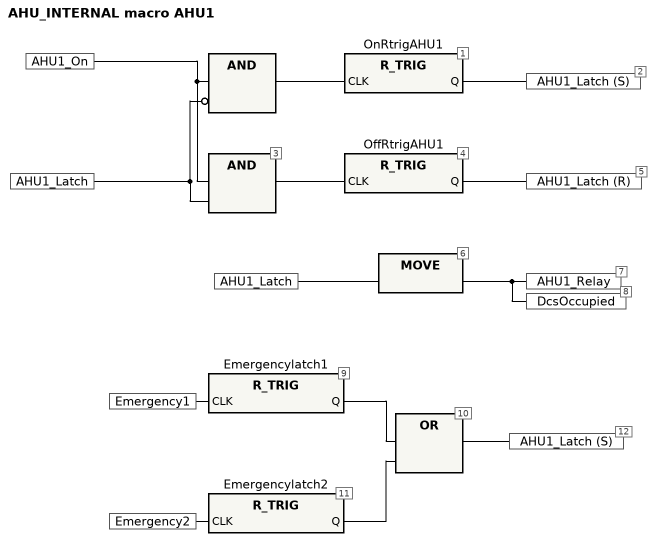
_CFC_ (* Continuous Function Chart, elements in execution order *)
#0 MACRO AHU1()
	#1 AND(AHU1_On, NOT AHU1_Latch)
	#2 OnRtrigAHU1:R_TRIG(CLK: #1)
	#3 S AHU1_Latch <= #2.Q
	#4 AND(AHU1_On, AHU1_Latch)
	#5 OffRtrigAHU1:R_TRIG(CLK: #4)
	#6 R AHU1_Latch <= #5.Q
	#7 MOVE(AHU1_Latch)
	#8 AHU1_Relay <= #7
	#9 DcsOccupied <= #7
	#10 Emergencylatch1:R_TRIG(CLK: Emergency1)
	#11 OR(#10.Q, #12.Q)
	#12 Emergencylatch2:R_TRIG(CLK: Emergency2)
	#13 S AHU1_Latch <= #11
END_MACRO
_END_CFC_
(* the same logic as Structured Text *)
(* macro AHU1 *)
OnRtrigAHU1(CLK := AHU1_On AND NOT AHU1_Latch);
IF OnRtrigAHU1.Q THEN AHU1_Latch := TRUE; END_IF;
OffRtrigAHU1(CLK := AHU1_On AND AHU1_Latch);
IF OffRtrigAHU1.Q THEN AHU1_Latch := FALSE; END_IF;
AHU1_Relay := AHU1_Latch;
DcsOccupied := AHU1_Latch;
Emergencylatch1(CLK := Emergency1);
_t232 := Emergencylatch1.Q OR Emergencylatch2.Q;
Emergencylatch2(CLK := Emergency2);
IF _t232 THEN AHU1_Latch := TRUE; END_IF;
END_FUNCTION_BLOCK

(* POU Module/ERROR_INTERNAL, CFC *)
FUNCTION_BLOCK ERROR_INTERNAL
VAR_INPUT
	status_error : BOOL;
	trip_error : BOOL;
END_VAR
VAR_OUTPUT
	Q:BOOL;
END_VAR
VAR
	ErrorFilter1: ErrorFilter;
END_VAR
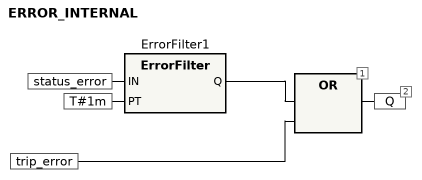
_CFC_ (* Continuous Function Chart, elements in execution order *)
#0 ErrorFilter1:ErrorFilter(IN: status_error, PT: T#1m)
#1 OR(#0.Q, trip_error)
#2 Q <= #1
_END_CFC_
(* the same logic as Structured Text *)
ErrorFilter1(IN := status_error, PT := T#1m);
Q := ErrorFilter1.Q OR trip_error;
END_FUNCTION_BLOCK

(* POU Module/ErrorFilter, ST *)
FUNCTION_BLOCK ErrorFilter
VAR_INPUT
	IN : BOOL;
	PT : TIME:=T#2s;
END_VAR
VAR_OUTPUT
	Q : BOOL;
END_VAR
VAR
	timer : TON;
END_VAR
IF PT <= T#0s THEN
	PT := T#2s;
END_IF

timer(IN:=IN , PT:=PT , Q=>Q );
END_FUNCTION_BLOCK

(* POU Module/Flowchart_7, CFC *)
FUNCTION_BLOCK Flowchart_7
VAR_IN_OUT
	Trigger : BOOL;
	Latch: BOOL;
END_VAR
VAR_OUTPUT
	DCS_Occupied: BOOL;
END_VAR
VAR
	DEV1: AHU_INTERNAL;
END_VAR
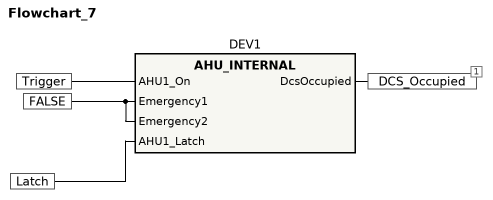
_CFC_ (* Continuous Function Chart, elements in execution order *)
#0 DEV1:AHU_INTERNAL(AHU1_On: Trigger, Emergency1: FALSE, Emergency2: FALSE, AHU1_Latch: Latch)
#1 DCS_Occupied <= #0.DcsOccupied
_END_CFC_
(* the same logic as Structured Text *)
DEV1(AHU1_On := Trigger, Emergency1 := FALSE, Emergency2 := FALSE, AHU1_Latch := Latch);
DCS_Occupied := DEV1.DcsOccupied;
END_FUNCTION_BLOCK

(* POU FieldAuxiliarryRoom1, ST *)
PROGRAM FieldAuxiliarryRoom1
VAR

	AHU_FAR1_common_alarm : BOOL;
	AHU_FAR1_dcs_occupied : BOOL;

	AHU_FAR1_dummy : BOOL;
	FB_AHU_FAR1: Flowchart_3_4_CTRL;

	AHU_FAR1_1_status AT%I* : BOOL;
	AHU_FAR1_1_trip AT%I* : BOOL;
	AHU_FAR1_1_mode AT%I* : BOOL;
	AHU_FAR1_1_belt AT%I* : BOOL;
	AHU_FAR1_1_fire AT%I* : BOOL;
	AHU_FAR1_1_gas AT%I* : BOOL;
	AHU_FAR1_1_smoke AT%I* : BOOL;

	AHU_FAR1_1_trigger : BOOL;
	AHU_FAR1_1_latch : BOOL;
	AHU_FAR1_1_common_alarm : BOOL;
	AHU_FAR1_1_status_error : BOOL;
	AHU_FAR1_1_trip_error : BOOL;
	AHU_FAR1_1_dcs_occupied : BOOL;

	AHU_FAR1_1_status_Filter : ErrorFilter;
	AHU_FAR1_1_trip_Filter : ErrorFilter;




	AHU_FAR1_2_status AT%I* : BOOL;
	AHU_FAR1_2_trip AT%I* : BOOL;
	AHU_FAR1_2_mode AT%I* : BOOL;
	AHU_FAR1_2_belt AT%I* : BOOL;
	AHU_FAR1_2_fire AT%I* : BOOL;
	AHU_FAR1_2_gas AT%I* : BOOL;
	AHU_FAR1_2_smoke AT%I* : BOOL;

	AHU_FAR1_2_trigger : BOOL;
	AHU_FAR1_2_latch : BOOL;
	AHU_FAR1_2_common_alarm : BOOL;
	AHU_FAR1_2_status_error : BOOL;
	AHU_FAR1_2_trip_error : BOOL;
	AHU_FAR1_2_dcs_occupied : BOOL;

	AHU_FAR1_2_status_Filter : ErrorFilter;
	AHU_FAR1_2_trip_Filter : ErrorFilter;

(***)


	EF_FAR1_common_alarm : BOOL;
	EF_FAR1_dcs_occupied : BOOL;

	EF_FAR1_dummy : BOOL;
	FB_EF_FAR1: Flowchart_3_4_CTRL;

	EF_FAR1_1A_status AT%I* : BOOL;
	EF_FAR1_1A_trip AT%I* : BOOL;
	EF_FAR1_1A_mode AT%I* : BOOL;

	EF_FAR1_1A_trigger : BOOL;
	EF_FAR1_1A_latch : BOOL;
	EF_FAR1_1A_common_alarm : BOOL;
	EF_FAR1_1A_status_error : BOOL;
	EF_FAR1_1A_trip_error : BOOL;
	EF_FAR1_1A_dcs_occupied : BOOL;

	EF_FAR1_1A_status_Filter : ErrorFilter;
	EF_FAR1_1A_trip_Filter : ErrorFilter;


	EF_FAR1_1B_status AT%I* : BOOL;
	EF_FAR1_1B_trip AT%I* : BOOL;
	EF_FAR1_1B_mode AT%I* : BOOL;

	EF_FAR1_1B_trigger : BOOL;
	EF_FAR1_1B_latch : BOOL;
	EF_FAR1_1B_common_alarm : BOOL;
	EF_FAR1_1B_status_error : BOOL;
	EF_FAR1_1B_trip_error : BOOL;
	EF_FAR1_1B_dcs_occupied : BOOL;

	EF_FAR1_1B_status_Filter : ErrorFilter;
	EF_FAR1_1B_trip_Filter : ErrorFilter;


(*********************)


	FB_EF_FAR1_3: Flowchart_7;

	EF_FAR1_3_status AT%I* : BOOL;
	EF_FAR1_3_trip AT%I* : BOOL;
	EF_FAR1_3_mode AT%I* : BOOL;

	EF_FAR1_3_trigger : BOOL;
	EF_FAR1_3_latch : BOOL;
	EF_FAR1_3_common_alarm : BOOL;
	EF_FAR1_3_status_error : BOOL;
	EF_FAR1_3_trip_error : BOOL;
	EF_FAR1_3_dcs_occupied : BOOL;

	EF_FAR1_3_status_Filter : ErrorFilter;
	EF_FAR1_3_trip_Filter : ErrorFilter;

(************************************)



	EF_FAR1_2_status AT%I* : BOOL;
	EF_FAR1_2_trip AT%I* : BOOL;
	EF_FAR1_2_mode AT%I* : BOOL;

	EF_FAR1_2_trigger : BOOL;
	EF_FAR1_2_latch : BOOL;
	EF_FAR1_2_common_alarm : BOOL;
	EF_FAR1_2_status_error : BOOL;
	EF_FAR1_2_trip_error : BOOL;
	EF_FAR1_2_dcs_occupied : BOOL;

	EF_FAR1_2_status_Filter : ErrorFilter;
	EF_FAR1_2_trip_Filter : ErrorFilter;

(*************************)

	FB_EDH_FAR1_1: Flowchart_5_6;
	EDH_FAR1_1_on_status : BOOL;
	EDH_FAR1_1_flow_status AT%I* : BOOL;
	EDH_FAR1_1_high_temp AT%I* : BOOL;

	EDH_FAR1_1_common_alarm : BOOL;
	EDH_FAR1_1_hightemp_error : BOOL;




(***************************)

	MD_FAR1_1A_damper_open AT%I* : BOOL;
	MD_FAR1_1A_damper_close AT%I* : BOOL;

	MD_FAR1_1B_damper_open AT%I* : BOOL;
	MD_FAR1_1B_damper_close AT%I* : BOOL;

	MD_FAR1_1C_damper_open AT%I* : BOOL;
	MD_FAR1_1C_damper_close AT%I* : BOOL;

	MD_EF_FAR1_2_damper_open AT%I* : BOOL;
	MD_EF_FAR1_2_damper_close AT%I* : BOOL;

(*************************)

	MFD_FAR1_1_damper_open AT%I* : BOOL;
	MFD_FAR1_1_damper_close AT%I* : BOOL;

	MFD_FAR1_2_damper_open AT%I* : BOOL;
	MFD_FAR1_2_damper_close AT%I* : BOOL;

	MFD_FAR1_3_damper_open AT%I* : BOOL;
	MFD_FAR1_3_damper_close AT%I* : BOOL;

	MFD_FAR1_4_damper_open AT%I* : BOOL;
	MFD_FAR1_4_damper_close AT%I* : BOOL;

	MFD_FAR1_5_damper_open AT%I* : BOOL;
	MFD_FAR1_5_damper_close AT%I* : BOOL;

	MFD_FAR1_6_damper_open AT%I* : BOOL;
	MFD_FAR1_6_damper_close AT%I* : BOOL;

(********************************)
	common_alarm AT%Q* : BOOL;
	dcs_occupied AT%Q* : BOOL;

END_VAR
AHU_FAR1_1_status_Filter(IN:=(NOT AHU_FAR1_1_status AND AHU_FAR1_1_latch),Q=>AHU_FAR1_1_status_error);
AHU_FAR1_1_trip_Filter(IN:=(AHU_FAR1_1_trip AND AHU_FAR1_1_latch),Q=>AHU_FAR1_1_trip_error);
AHU_FAR1_1_common_alarm := AHU_FAR1_1_fire OR AHU_FAR1_1_gas OR AHU_FAR1_1_smoke OR AHU_FAR1_1_status_error OR AHU_FAR1_1_trip_error;


AHU_FAR1_2_status_Filter(IN:=(NOT AHU_FAR1_2_status AND AHU_FAR1_2_latch),Q=>AHU_FAR1_2_status_error);
AHU_FAR1_2_trip_Filter(IN:=(AHU_FAR1_2_trip AND AHU_FAR1_2_latch),Q=>AHU_FAR1_2_trip_error);
AHU_FAR1_2_common_alarm := AHU_FAR1_2_fire OR AHU_FAR1_2_gas OR AHU_FAR1_2_smoke OR AHU_FAR1_2_status_error OR AHU_FAR1_2_trip_error;


AHU_FAR1_common_alarm := AHU_FAR1_1_common_alarm OR AHU_FAR1_2_common_alarm ;
AHU_FAR1_dcs_occupied := AHU_FAR1_1_dcs_occupied OR AHU_FAR1_2_dcs_occupied;

	FB_AHU_FAR1(
	ON1:=AHU_FAR1_1_trigger ,
	ON2:=AHU_FAR1_2_trigger ,
	ON3:=FALSE ,
	status_error_1:= AHU_FAR1_1_status_error,
	status_error_2:=AHU_FAR1_2_status_error ,
	status_error_3:=FALSE ,
	trip_error_1:=AHU_FAR1_1_trip_error ,
	trip_error_2:=AHU_FAR1_2_trip_error ,
	trip_error_3:=FALSE ,
	Latch1:=AHU_FAR1_1_latch ,
	Latch2:=AHU_FAR1_2_latch ,
	Latch3:=AHU_FAR1_dummy ,
	DcsOccupied_1=>AHU_FAR1_1_dcs_occupied ,
	DcsOccupied_2=>AHU_FAR1_2_dcs_occupied ,
	DcsOccupied_3=> );


EF_FAR1_1A_status_Filter(IN:=(NOT EF_FAR1_1A_status AND EF_FAR1_1A_latch),Q=>EF_FAR1_1A_status_error);
EF_FAR1_1A_trip_Filter(IN:=(EF_FAR1_1A_trip AND EF_FAR1_1A_latch),Q=>EF_FAR1_1A_trip_error);
EF_FAR1_1A_common_alarm := EF_FAR1_1A_status_error OR EF_FAR1_1A_trip_error;



EF_FAR1_1B_status_Filter(IN:=(NOT EF_FAR1_1B_status AND EF_FAR1_1B_latch),Q=>EF_FAR1_1B_status_error);
EF_FAR1_1B_trip_Filter(IN:=(EF_FAR1_1B_trip AND EF_FAR1_1B_latch),Q=>EF_FAR1_1B_trip_error);
EF_FAR1_1B_common_alarm := EF_FAR1_1B_status_error OR EF_FAR1_1B_trip_error;


EF_FAR1_common_alarm := EF_FAR1_1A_common_alarm OR EF_FAR1_1B_common_alarm;
EF_FAR1_dcs_occupied := EF_FAR1_1A_dcs_occupied OR EF_FAR1_1B_dcs_occupied;

	FB_EF_FAR1(
	ON1:=EF_FAR1_1A_trigger ,
	ON2:=EF_FAR1_1B_trigger ,
	ON3:=FALSE ,
	status_error_1:= EF_FAR1_1A_status_error,
	status_error_2:=EF_FAR1_1B_status_error ,
	status_error_3:=FALSE ,
	trip_error_1:=EF_FAR1_1A_trip_error ,
	trip_error_2:=EF_FAR1_1B_trip_error ,
	trip_error_3:=FALSE ,
	Latch1:=EF_FAR1_1A_latch ,
	Latch2:=EF_FAR1_1B_latch ,
	Latch3:=EF_FAR1_dummy ,
	DcsOccupied_1=>EF_FAR1_1A_dcs_occupied ,
	DcsOccupied_2=>EF_FAR1_1B_dcs_occupied ,
	DcsOccupied_3=> );


(**************************)

EF_FAR1_3_status_Filter(IN:=(NOT EF_FAR1_3_status AND EF_FAR1_3_latch),Q=>EF_FAR1_3_status_error);
EF_FAR1_3_trip_Filter(IN:=(EF_FAR1_3_trip AND EF_FAR1_3_latch),Q=>EF_FAR1_3_trip_error);
EF_FAR1_3_common_alarm := EF_FAR1_3_status_error OR EF_FAR1_3_trip_error;


FB_EF_FAR1_3(
Trigger:=EF_FAR1_3_trigger ,
Latch:=EF_FAR1_3_latch ,
DCS_Occupied=>EF_FAR1_3_dcs_occupied );


(*************************)


EF_FAR1_2_status_Filter(IN:=(NOT EF_FAR1_2_status AND EF_FAR1_2_latch),Q=>EF_FAR1_2_status_error);
EF_FAR1_2_trip_Filter(IN:=(EF_FAR1_2_trip AND EF_FAR1_2_latch),Q=>EF_FAR1_2_trip_error);
EF_FAR1_2_common_alarm := EF_FAR1_2_status_error OR EF_FAR1_2_trip_error;


(***************************)

EDH_FAR1_1_on_status := AHU_FAR1_dcs_occupied;

FB_EDH_FAR1_1(on_status:= EDH_FAR1_1_on_status , flow_status:= EDH_FAR1_1_flow_status , high_temp:= EDH_FAR1_1_high_temp);

EDH_FAR1_1_hightemp_error := EDH_FAR1_1_high_temp;
EDH_FAR1_1_common_alarm := EDH_FAR1_1_hightemp_error;


(***************************)

common_alarm := AHU_FAR1_common_alarm OR EF_FAR1_common_alarm OR EF_FAR1_3_common_alarm OR EF_FAR1_2_common_alarm;

dcs_occupied := AHU_FAR1_dcs_occupied OR EF_FAR1_dcs_occupied OR EF_FAR1_3_dcs_occupied;
END_PROGRAM

(* POU CCB_GroundFloor, ST *)
PROGRAM CCB_GroundFloor
VAR

	AHU_CCBG_01_status AT%I* : BOOL;
	AHU_CCBG_01_trip AT%I* : BOOL;
	AHU_CCBG_01_mode AT%I* : BOOL;
	AHU_CCBG_01_belt AT%I* : BOOL;
	AHU_CCBG_01_fire AT%I* : BOOL;
	AHU_CCBG_01_gas AT%I* : BOOL;
	AHU_CCBG_01_smoke AT%I* : BOOL;

	AHU_CCBG_01_trigger : BOOL;
	AHU_CCBG_01_latch : BOOL;
	AHU_CCBG_01_common_alarm : BOOL;
	AHU_CCBG_01_status_error : BOOL;
	AHU_CCBG_01_trip_error : BOOL;
	AHU_CCBG_01_dcs_occupied : BOOL;

	AHU_CCBG_01_status_Filter : ErrorFilter;
	AHU_CCBG_01_trip_Filter : ErrorFilter;



	AHU_CCBG_02_status AT%I* : BOOL;
	AHU_CCBG_02_trip AT%I* : BOOL;
	AHU_CCBG_02_mode AT%I* : BOOL;
	AHU_CCBG_02_belt AT%I* : BOOL;
	AHU_CCBG_02_fire AT%I* : BOOL;
	AHU_CCBG_02_gas AT%I* : BOOL;
	AHU_CCBG_02_smoke AT%I* : BOOL;

	AHU_CCBG_02_trigger : BOOL;
	AHU_CCBG_02_latch : BOOL;
	AHU_CCBG_02_common_alarm : BOOL;
	AHU_CCBG_02_status_error : BOOL;
	AHU_CCBG_02_trip_error : BOOL;
	AHU_CCBG_02_dcs_occupied : BOOL;

	AHU_CCBG_02_status_Filter : ErrorFilter;
	AHU_CCBG_02_trip_Filter : ErrorFilter;



	AHU_CCBG_03_status AT%I* : BOOL;
	AHU_CCBG_03_trip AT%I* : BOOL;
	AHU_CCBG_03_mode AT%I* : BOOL;
	AHU_CCBG_03_belt AT%I* : BOOL;
	AHU_CCBG_03_fire AT%I* : BOOL;
	AHU_CCBG_03_gas AT%I* : BOOL;
	AHU_CCBG_03_smoke AT%I* : BOOL;

	AHU_CCBG_03_trigger : BOOL;
	AHU_CCBG_03_latch : BOOL;
	AHU_CCBG_03_common_alarm : BOOL;
	AHU_CCBG_03_status_error : BOOL;
	AHU_CCBG_03_trip_error : BOOL;
	AHU_CCBG_03_dcs_occupied : BOOL;

	AHU_CCBG_03_status_Filter : ErrorFilter;
	AHU_CCBG_03_trip_Filter : ErrorFilter;

	AHU_CCCBG :Flowchart_1_2_CTRL;

(******************************************************************************************************)

	EF_CCB_1_status AT%I* : BOOL;
	EF_CCB_1_trip AT%I* : BOOL;
	EF_CCB_1_mode AT%I* : BOOL;

	EF_CCB_1_trigger : BOOL;
	EF_CCB_1_latch : BOOL;
	EF_CCB_1_common_alarm : BOOL;
	EF_CCB_1_status_error : BOOL;
	EF_CCB_1_trip_error : BOOL;
	EF_CCB_1_dcs_occupied : BOOL;

	EF_CCB_1_status_Filter : ErrorFilter;
	EF_CCB_1_trip_Filter : ErrorFilter;

	EF_CCB_2_status AT%I* : BOOL;
	EF_CCB_2_trip AT%I* : BOOL;
	EF_CCB_2_mode AT%I* : BOOL;

	EF_CCB_2_trigger : BOOL;
	EF_CCB_2_latch : BOOL;
	EF_CCB_2_common_alarm : BOOL;
	EF_CCB_2_status_error : BOOL;
	EF_CCB_2_trip_error : BOOL;
	EF_CCB_2_dcs_occupied : BOOL;

	EF_CCB_2_status_Filter : ErrorFilter;
	EF_CCB_2_trip_Filter : ErrorFilter;

	EF_CCB :Flowchart_3_4_CTRL;
	EF_CCB_Dummy: BOOL;

(********************************************************************************************************************************************************)

	TEF_CCB_01_status AT%I* : BOOL;
	TEF_CCB_01_trip AT%I* : BOOL;
	TEF_CCB_01_mode AT%I* : BOOL;

	TEF_CCB_01_trigger : BOOL;
	TEF_CCB_01_latch : BOOL;
	TEF_CCB_01_common_alarm : BOOL;
	TEF_CCB_01_status_error : BOOL;
	TEF_CCB_01_trip_error : BOOL;
	TEF_CCB_01_dcs_occupied : BOOL;

	TEF_CCB_01_status_Filter : ErrorFilter;
	TEF_CCB_01_trip_Filter : ErrorFilter;

	TEC_CCB :Flowchart_7;


(***************************************************************************************************************************************************)

	EF_CCB_7A_status AT%I* : BOOL;
	EF_CCB_7A_trip AT%I* : BOOL;

	EF_CCB_7A_common_alarm : BOOL;
	EF_CCB_7A_status_error : BOOL;
	EF_CCB_7A_trip_error : BOOL;

	EF_CCB_7A_status_Filter : ErrorFilter;
	EF_CCB_7A_trip_Filter : ErrorFilter;


	EF_CCB_7B_status AT%I* : BOOL;
	EF_CCB_7B_trip AT%I* : BOOL;

	EF_CCB_7B_trigger : BOOL;
	EF_CCB_7B_latch : BOOL;
	EF_CCB_7B_common_alarm : BOOL;
	EF_CCB_7B_status_error : BOOL;
	EF_CCB_7B_trip_error : BOOL;
	EF_CCB_7B_dcs_occupied : BOOL;

	EF_CCB_7B_status_Filter : ErrorFilter;
	EF_CCB_7B_trip_Filter : ErrorFilter;

	EF_CCB_08_status AT%I* : BOOL;
	EF_CCB_08_trip AT%I* : BOOL;

	EF_CCB_08_trigger : BOOL;
	EF_CCB_08_latch : BOOL;
	EF_CCB_08_common_alarm : BOOL;
	EF_CCB_08_status_error : BOOL;
	EF_CCB_08_trip_error : BOOL;
	EF_CCB_08_dcs_occupied : BOOL;

	EF_CCB_08_status_Filter : ErrorFilter;
	EF_CCB_08_trip_Filter : ErrorFilter;

(******************************************************************************************************************************)

	EH_CCB_01_on_status  : BOOL;
	EH_CCB_01_flow_status AT%I* : BOOL;
	EH_CCB_01_high_temp AT%I* : BOOL;

	EH_CCB_01_common_alarm : BOOL;
	EH_CCB_01_hightemp_error : BOOL;

	EH_CCB_01_FB :Flowchart_5_6;



	EH_CCB_02_on_status  : BOOL;
	EH_CCB_02_flow_status AT%I* : BOOL;
	EH_CCB_02_high_temp AT%I* : BOOL;

	EH_CCB_02_common_alarm : BOOL;
	EH_CCB_02_hightemp_error : BOOL;

	EH_CCB_02_FB :Flowchart_5_6;

(******************************************************************************************************************************)

	MD_CCBG_1_damper_open AT%I* : BOOL;
	MD_CCBG_1_damper_close AT%I* : BOOL;
	MD_CCBG_2_damper_open AT%I* : BOOL;
	MD_CCBG_2_damper_close AT%I* : BOOL;
	MD_CCBG_3_damper_open AT%I* : BOOL;
	MD_CCBG_3_damper_close AT%I* : BOOL;
	MD_CCBG_4_damper_open AT%I* : BOOL;
	MD_CCBG_4_damper_close AT%I* : BOOL;

	MD_EF_CCB_7A_damper_open AT%I* : BOOL;
	MD_EF_CCB_7A_damper_close AT%I* : BOOL;
	MD_EF_CCB_7B_damper_open AT%I* : BOOL;
	MD_EF_CCB_7B_damper_close AT%I* : BOOL;
	MD_EF_CCB_8_damper_open AT%I* : BOOL;
	MD_EF_CCB_8_damper_close AT%I* : BOOL;

(***************************************************************************************************************************)

	MFD_CCB_1_damper_open AT%I* : BOOL;
	MFD_CCB_1_damper_close AT%I* : BOOL;
	MFD_CCB_2_damper_open AT%I* : BOOL;
	MFD_CCB_2_damper_close AT%I* : BOOL;
	MFD_CCB_3_damper_open AT%I* : BOOL;
	MFD_CCB_3_damper_close AT%I* : BOOL;
	MFD_CCB_4_damper_open AT%I* : BOOL;
	MFD_CCB_4_damper_close AT%I* : BOOL;
	MFD_CCB_5_damper_open AT%I* : BOOL;
	MFD_CCB_5_damper_close AT%I* : BOOL;
	MFD_CCB_6_damper_open AT%I* : BOOL;
	MFD_CCB_6_damper_close AT%I* : BOOL;
	MFD_CCB_7_damper_open AT%I* : BOOL;
	MFD_CCB_7_damper_close AT%I* : BOOL;
	MFD_CCB_8_damper_open AT%I* : BOOL;
	MFD_CCB_8_damper_close AT%I* : BOOL;
	MFD_CCB_9_damper_open AT%I* : BOOL;
	MFD_CCB_9_damper_close AT%I* : BOOL;
	MFD_CCB_10_damper_open AT%I* : BOOL;
	MFD_CCB_10_damper_close AT%I* : BOOL;

	DCS_Occupied AT%Q*: BOOL;
	common_alarm AT %Q*: BOOL;
END_VAR
AHU_CCBG_01_status_Filter(IN:=(NOT AHU_CCBG_01_status AND AHU_CCBG_01_latch),Q=>AHU_CCBG_01_status_error);
AHU_CCBG_01_trip_Filter(IN:=(AHU_CCBG_01_trip AND AHU_CCBG_01_latch),Q=>AHU_CCBG_01_trip_error);
AHU_CCBG_01_common_alarm := AHU_CCBG_01_fire OR AHU_CCBG_01_gas OR AHU_CCBG_01_smoke OR AHU_CCBG_01_status_error OR AHU_CCBG_01_trip_error;

AHU_CCBG_02_status_Filter(IN:=(NOT AHU_CCBG_02_status AND AHU_CCBG_02_latch),Q=>AHU_CCBG_02_status_error);
AHU_CCBG_02_trip_Filter(IN:=(AHU_CCBG_02_trip AND AHU_CCBG_02_latch),Q=>AHU_CCBG_02_trip_error);
AHU_CCBG_02_common_alarm := AHU_CCBG_02_fire OR AHU_CCBG_02_gas OR AHU_CCBG_02_smoke OR AHU_CCBG_02_status_error OR AHU_CCBG_02_trip_error;

AHU_CCBG_03_status_Filter(IN:=(NOT AHU_CCBG_03_status AND AHU_CCBG_03_latch),Q=>AHU_CCBG_03_status_error);
AHU_CCBG_03_trip_Filter(IN:=(AHU_CCBG_03_trip AND AHU_CCBG_03_latch),Q=>AHU_CCBG_03_trip_error);
AHU_CCBG_02_common_alarm := AHU_CCBG_02_fire OR AHU_CCBG_02_gas OR AHU_CCBG_02_smoke OR AHU_CCBG_02_status_error OR AHU_CCBG_02_trip_error;

AHU_CCCBG(
	ON1:=AHU_CCBG_01_trigger ,
	ON2:=AHU_CCBG_02_trigger ,
	ON3:=AHU_CCBG_03_trigger ,
	status_error_1:= AHU_CCBG_01_status_error,
	status_error_2:=AHU_CCBG_02_status_error ,
	status_error_3:=AHU_CCBG_03_status_error ,
	trip_error_1:=AHU_CCBG_01_trip_error ,
	trip_error_2:=AHU_CCBG_02_trip_error ,
	trip_error_3:=AHU_CCBG_03_trip_error ,
	Latch1:=AHU_CCBG_01_latch ,
	Latch2:=AHU_CCBG_02_latch ,
	Latch3:=AHU_CCBG_03_latch ,
	DcsOccupied_1=>AHU_CCBG_01_dcs_occupied ,
	DcsOccupied_2=>AHU_CCBG_02_dcs_occupied ,
	DcsOccupied_3=>AHU_CCBG_03_dcs_occupied );

(***********************************************************************************************************************************************************************************************)

EF_CCB_1_status_Filter(IN:=(NOT EF_CCB_1_status AND EF_CCB_1_latch),Q=>EF_CCB_1_status_error);
EF_CCB_1_trip_Filter(IN:=(EF_CCB_1_trip AND EF_CCB_1_latch),Q=>EF_CCB_1_trip_error);
EF_CCB_1_common_alarm := EF_CCB_1_status_error OR EF_CCB_1_trip_error;

EF_CCB_2_status_Filter(IN:=(NOT EF_CCB_2_status AND EF_CCB_2_latch),Q=>EF_CCB_2_status_error);
EF_CCB_2_trip_Filter(IN:=(EF_CCB_2_trip AND EF_CCB_2_latch),Q=>EF_CCB_2_trip_error);
EF_CCB_2_common_alarm := EF_CCB_2_status_error OR EF_CCB_2_trip_error;

EF_CCB(
	ON1:=EF_CCB_1_trigger ,
	ON2:=EF_CCB_2_trigger ,
	ON3:=FALSE ,
	status_error_1:= EF_CCB_2_status_error,
	status_error_2:=EF_CCB_2_status_error,
	status_error_3:=FALSE ,
	trip_error_1:=EF_CCB_1_trip_error ,
	trip_error_2:=EF_CCB_2_trip_error ,
	trip_error_3:= FALSE,
	Latch1:=EF_CCB_1_latch ,
	Latch2:= EF_CCB_2_latch,
	Latch3:=EF_CCB_Dummy ,
	DcsOccupied_1=>EF_CCB_1_dcs_occupied ,
	DcsOccupied_2=>EF_CCB_2_dcs_occupied ,
	DcsOccupied_3=> );

(*******************************************************************************************************************************)

TEF_CCB_01_status_Filter(IN:=(NOT TEF_CCB_01_status AND TEF_CCB_01_latch),Q=>TEF_CCB_01_status_error);
TEF_CCB_01_trip_Filter(IN:=(TEF_CCB_01_trip AND TEF_CCB_01_latch),Q=>TEF_CCB_01_trip_error);
TEF_CCB_01_common_alarm := TEF_CCB_01_status_error OR TEF_CCB_01_trip_error;

TEC_CCB(
	Trigger:=TEF_CCB_01_trigger ,
	Latch:=TEF_CCB_01_latch ,
	DCS_Occupied=>TEF_CCB_01_dcs_occupied );
(*******************************************************************************************************************************)


EF_CCB_7A_status_Filter(IN:=(NOT EF_CCB_7A_status),Q=>EF_CCB_7A_status_error);
EF_CCB_7A_trip_Filter(IN:=(EF_CCB_7A_trip),Q=>EF_CCB_7A_trip_error);
EF_CCB_7A_common_alarm := EF_CCB_7A_status_error OR EF_CCB_7A_trip_error;

EF_CCB_7B_status_Filter(IN:=(NOT EF_CCB_7B_status),Q=>EF_CCB_7B_status_error);
EF_CCB_7B_trip_Filter(IN:=(EF_CCB_7B_trip),Q=>EF_CCB_7B_trip_error);
EF_CCB_7B_common_alarm := EF_CCB_7B_status_error OR EF_CCB_7B_trip_error;

EF_CCB_08_status_Filter(IN:=(NOT EF_CCB_08_status),Q=>EF_CCB_08_status_error);
EF_CCB_08_trip_Filter(IN:=(EF_CCB_08_trip),Q=>EF_CCB_08_trip_error);
EF_CCB_08_common_alarm := EF_CCB_08_status_error OR EF_CCB_08_trip_error;


(******************************************************************************************************************************)


EH_CCB_01_on_status := AHU_CCBG_01_dcs_occupied OR AHU_CCBG_02_dcs_occupied OR AHU_CCBG_03_dcs_occupied;
EH_CCB_01_hightemp_error := EH_CCB_01_high_temp;
EH_CCB_01_common_alarm := EH_CCB_01_hightemp_error;

EH_CCB_01_FB(on_status:= EH_CCB_01_on_status , flow_status:= EH_CCB_01_flow_status , high_temp:= EH_CCB_01_high_temp);


EH_CCB_02_on_status := AHU_CCBG_01_dcs_occupied OR AHU_CCBG_02_dcs_occupied OR AHU_CCBG_03_dcs_occupied;
EH_CCB_02_hightemp_error := EH_CCB_02_high_temp;
EH_CCB_02_common_alarm := EH_CCB_02_hightemp_error;

EH_CCB_02_FB(on_status:=EH_CCB_02_on_status , flow_status:=EH_CCB_02_flow_status , high_temp:=EH_CCB_02_high_temp );


(******************************************************************************************************************************)


DCS_Occupied := AHU_CCBG_01_dcs_occupied OR AHU_CCBG_02_dcs_occupied OR AHU_CCBG_03_dcs_occupied OR EF_CCB_1_dcs_occupied OR EF_CCB_2_dcs_occupied OR TEF_CCB_01_dcs_occupied;
common_alarm := AHU_CCBG_01_common_alarm OR AHU_CCBG_02_common_alarm OR AHU_CCBG_03_common_alarm OR EF_CCB_1_common_alarm OR EF_CCB_2_common_alarm OR TEF_CCB_01_common_alarm OR EF_CCB_7A_common_alarm OR EF_CCB_7B_common_alarm OR EF_CCB_08_common_alarm OR EH_CCB_01_common_alarm OR EH_CCB_02_common_alarm;
END_PROGRAM

(* POU Module/Flowchart_1_2_CTRL, CFC *)
FUNCTION_BLOCK Flowchart_1_2_CTRL
VAR
	DEV_1: AHU_INTERNAL;
	DEV_2: AHU_INTERNAL;
	DEV_3: AHU_INTERNAL;

	DEV1_ErrorInternal_1: ERROR_INTERNAL;
	DEV1_ErrorInternal_2: ERROR_INTERNAL;

	DEV2_ErrorInternal_1: ERROR_INTERNAL;
	DEV2_ErrorInternal_2: ERROR_INTERNAL;

	DEV3_ErrorInternal_1: ERROR_INTERNAL;
	DEV3_ErrorInternal_2: ERROR_INTERNAL;
END_VAR
VAR_INPUT
	ON1: BOOL;
	ON2: BOOL;
	ON3: BOOL;

	status_error_1 : BOOL;
	status_error_2 : BOOL;
	status_error_3 : BOOL;

	trip_error_1 : BOOL;
	trip_error_2 : BOOL;
	trip_error_3 : BOOL;


END_VAR
VAR_IN_OUT
	Latch1:BOOL;
	Latch2:BOOL;
	Latch3:BOOL;
END_VAR
VAR_OUTPUT
	DcsOccupied_1: BOOL;
	DcsOccupied_2: BOOL;
	DcsOccupied_3: BOOL;
END_VAR
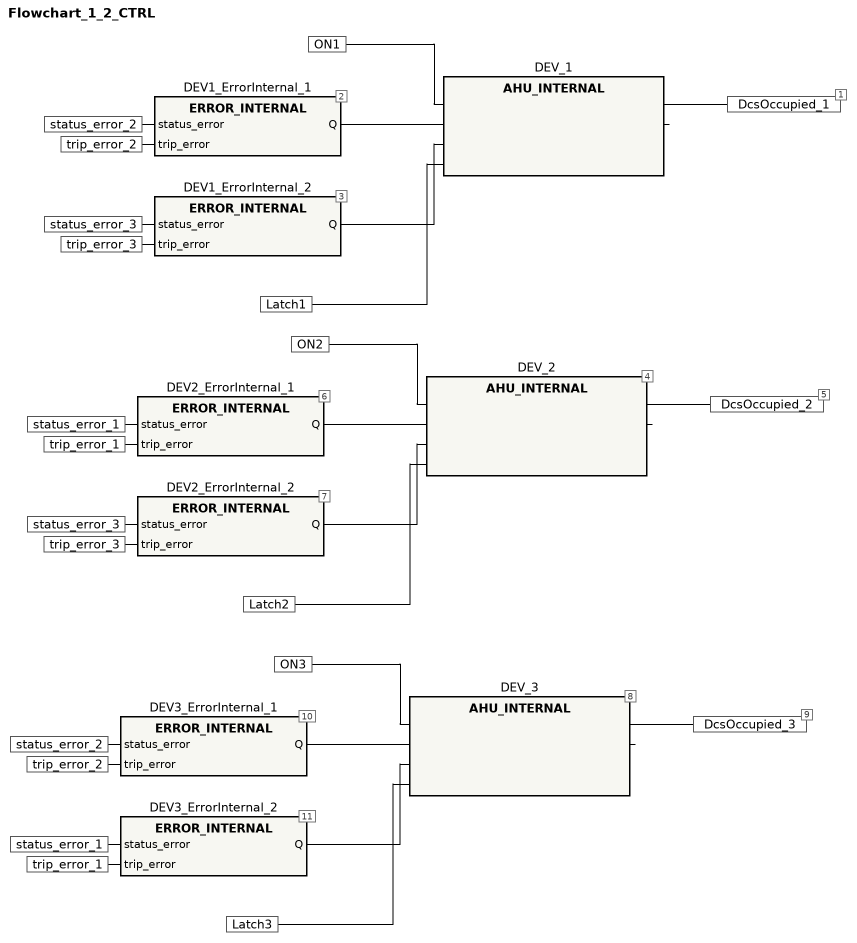
_CFC_ (* Continuous Function Chart, elements in execution order *)
#0 DEV_1:AHU_INTERNAL(ON1, #2.Q, #3.Q, Latch1)
#1 DcsOccupied_1 <= #0.out 1
#2 DEV1_ErrorInternal_1:ERROR_INTERNAL(status_error: status_error_2, trip_error: trip_error_2)
#3 DEV1_ErrorInternal_2:ERROR_INTERNAL(status_error: status_error_3, trip_error: trip_error_3)
#4 DEV_2:AHU_INTERNAL(ON2, #6.Q, #7.Q, Latch2)
#5 DcsOccupied_2 <= #4.out 1
#6 DEV2_ErrorInternal_1:ERROR_INTERNAL(status_error: status_error_1, trip_error: trip_error_1)
#7 DEV2_ErrorInternal_2:ERROR_INTERNAL(status_error: status_error_3, trip_error: trip_error_3)
#8 DEV_3:AHU_INTERNAL(ON3, #10.Q, #11.Q, Latch3)
#9 DcsOccupied_3 <= #8.out 1
#10 DEV3_ErrorInternal_1:ERROR_INTERNAL(status_error: status_error_2, trip_error: trip_error_2)
#11 DEV3_ErrorInternal_2:ERROR_INTERNAL(status_error: status_error_1, trip_error: trip_error_1)
_END_CFC_
END_FUNCTION_BLOCK

(* POU CCB_FirstFloor, ST *)
PROGRAM CCB_FirstFloor
VAR

	FCU_CCB1_23A_status AT%I* : BOOL;
	FCU_CCB1_23A_trip AT%I* : BOOL;
	FCU_CCB1_23A_mode AT%I* : BOOL;

	FCU_CCB1_23A_trigger : BOOL;
	FCU_CCB1_23A_latch : BOOL;
	FCU_CCB1_23A_common_alarm : BOOL;
	FCU_CCB1_23A_status_error : BOOL;
	FCU_CCB1_23A_trip_error : BOOL;
	FCU_CCB1_23A_dcs_occupied : BOOL;

	FCU_CCB1_23A_status_Filter : ErrorFilter;
	FCU_CCB1_23A_trip_Filter : ErrorFilter;

	FCU_CCB1_23A_FB :Flowchart_7;


(*************************************************************************************************************)


	FCU_CCB1_23B_status AT%I* : BOOL;
	FCU_CCB1_23B_trip AT%I* : BOOL;
	FCU_CCB1_23B_mode AT%I* : BOOL;

	FCU_CCB1_23B_trigger : BOOL;
	FCU_CCB1_23B_latch : BOOL;
	FCU_CCB1_23B_common_alarm : BOOL;
	FCU_CCB1_23B_status_error : BOOL;
	FCU_CCB1_23B_trip_error : BOOL;
	FCU_CCB1_23B_dcs_occupied : BOOL;

	FCU_CCB1_23B_status_Filter : ErrorFilter;
	FCU_CCB1_23B_trip_Filter : ErrorFilter;

	FCU_CCB1_23B_FB :Flowchart_7;


(*************************************************************************************************************)


	FCU_CCB1_23C_status AT%I* : BOOL;
	FCU_CCB1_23C_trip AT%I* : BOOL;
	FCU_CCB1_23C_mode AT%I* : BOOL;

	FCU_CCB1_23C_trigger : BOOL;
	FCU_CCB1_23C_latch : BOOL;
	FCU_CCB1_23C_common_alarm : BOOL;
	FCU_CCB1_23C_status_error : BOOL;
	FCU_CCB1_23C_trip_error : BOOL;
	FCU_CCB1_23C_dcs_occupied : BOOL;

	FCU_CCB1_23C_status_Filter : ErrorFilter;
	FCU_CCB1_23C_trip_Filter : ErrorFilter;

	FCU_CCB1_23C_FB :Flowchart_7;


	DCS_Occupied AT %Q*: BOOL;
	common_alarm AT %Q*: BOOL;
END_VAR
FCU_CCB1_23A_status_Filter(IN:=(NOT FCU_CCB1_23A_status AND FCU_CCB1_23A_latch),Q=>FCU_CCB1_23A_status_error);
FCU_CCB1_23A_trip_Filter(IN:=(FCU_CCB1_23A_trip AND FCU_CCB1_23A_latch),Q=>FCU_CCB1_23A_trip_error);
FCU_CCB1_23A_common_alarm := FCU_CCB1_23A_status_error OR FCU_CCB1_23A_trip_error;

FCU_CCB1_23A_FB(
	Trigger:=FCU_CCB1_23A_trigger ,
	Latch:= FCU_CCB1_23A_latch,
	DCS_Occupied=>FCU_CCB1_23A_dcs_occupied );


(*************************************************************************************************************)


FCU_CCB1_23B_status_Filter(IN:=(NOT FCU_CCB1_23B_status AND FCU_CCB1_23B_latch),Q=>FCU_CCB1_23B_status_error);
FCU_CCB1_23B_trip_Filter(IN:=(FCU_CCB1_23B_trip AND FCU_CCB1_23B_latch),Q=>FCU_CCB1_23B_trip_error);
FCU_CCB1_23B_common_alarm := FCU_CCB1_23B_status_error OR FCU_CCB1_23B_trip_error;

FCU_CCB1_23B_FB(
	Trigger:=FCU_CCB1_23B_trigger ,
	Latch:= FCU_CCB1_23B_latch,
	DCS_Occupied=>FCU_CCB1_23B_dcs_occupied );

(*************************************************************************************************************)

FCU_CCB1_23C_status_Filter(IN:=(NOT FCU_CCB1_23C_status AND FCU_CCB1_23C_latch),Q=>FCU_CCB1_23C_status_error);
FCU_CCB1_23C_trip_Filter(IN:=(FCU_CCB1_23C_trip AND FCU_CCB1_23C_latch),Q=>FCU_CCB1_23C_trip_error);
FCU_CCB1_23C_common_alarm := FCU_CCB1_23C_status_error OR FCU_CCB1_23C_trip_error;

FCU_CCB1_23C_FB(
	Trigger:=FCU_CCB1_23C_trigger ,
	Latch:= FCU_CCB1_23C_latch,
	DCS_Occupied=>FCU_CCB1_23C_dcs_occupied );


(*************************************************************************************************************)


DCS_Occupied := FCU_CCB1_23A_dcs_occupied OR FCU_CCB1_23B_dcs_occupied OR FCU_CCB1_23C_dcs_occupied;
common_alarm := FCU_CCB1_23A_common_alarm OR FCU_CCB1_23B_common_alarm OR FCU_CCB1_23C_common_alarm;
END_PROGRAM

(* POU AmmoniaUreaSubstation, ST *)
PROGRAM AmmoniaUreaSubstation
VAR
	AHU_AUSS_common_alarm : BOOL;
	AHU_AUSS_dcs_occupied : BOOL;

	AHU_AUSS_dummy : BOOL;
	FB_AHU_AUSS: Flowchart_3_4_CTRL;

	AHU_AUSS_1_status AT%I* : BOOL;
	AHU_AUSS_1_trip AT%I* : BOOL;
	AHU_AUSS_1_mode AT%I* : BOOL;
	AHU_AUSS_1_belt AT%I* : BOOL;
	AHU_AUSS_1_fire AT%I* : BOOL;
	AHU_AUSS_1_gas AT%I* : BOOL;
	AHU_AUSS_1_smoke AT%I* : BOOL;

	AHU_AUSS_1_trigger : BOOL;
	AHU_AUSS_1_latch : BOOL;
	AHU_AUSS_1_common_alarm : BOOL;
	AHU_AUSS_1_status_error : BOOL;
	AHU_AUSS_1_trip_error : BOOL;
	AHU_AUSS_1_dcs_occupied : BOOL;

	AHU_AUSS_1_status_Filter : ErrorFilter;
	AHU_AUSS_1_trip_Filter : ErrorFilter;


	AHU_AUSS_2_status AT%I* : BOOL;
	AHU_AUSS_2_trip AT%I* : BOOL;
	AHU_AUSS_2_mode AT%I* : BOOL;
	AHU_AUSS_2_belt AT%I* : BOOL;
	AHU_AUSS_2_fire AT%I* : BOOL;
	AHU_AUSS_2_gas AT%I* : BOOL;
	AHU_AUSS_2_smoke AT%I* : BOOL;

	AHU_AUSS_2_trigger : BOOL;
	AHU_AUSS_2_latch : BOOL;
	AHU_AUSS_2_common_alarm : BOOL;
	AHU_AUSS_2_status_error : BOOL;
	AHU_AUSS_2_trip_error : BOOL;
	AHU_AUSS_2_dcs_occupied : BOOL;

	AHU_AUSS_2_status_Filter : ErrorFilter;
	AHU_AUSS_2_trip_Filter : ErrorFilter;



(*****************************)


	EF_AUSS_common_alarm : BOOL;
	EF_AUSS_dcs_occupied : BOOL;

	EF_AUSS_dummy : BOOL;
	FB_EF_AUSS: Flowchart_3_4_CTRL;

	EF_AUSS_1_status AT%I* : BOOL;
	EF_AUSS_1_trip AT%I* : BOOL;
	EF_AUSS_1_mode AT%I* : BOOL;

	EF_AUSS_1_trigger : BOOL;
	EF_AUSS_1_latch : BOOL;
	EF_AUSS_1_common_alarm : BOOL;
	EF_AUSS_1_status_error : BOOL;
	EF_AUSS_1_trip_error : BOOL;
	EF_AUSS_1_dcs_occupied : BOOL;

	EF_AUSS_1_status_Filter : ErrorFilter;
	EF_AUSS_1_trip_Filter : ErrorFilter;


	EF_AUSS_2_status AT%I* : BOOL;
	EF_AUSS_2_trip AT%I* : BOOL;
	EF_AUSS_2_mode AT%I* : BOOL;

	EF_AUSS_2_trigger : BOOL;
	EF_AUSS_2_latch : BOOL;
	EF_AUSS_2_common_alarm : BOOL;
	EF_AUSS_2_status_error : BOOL;
	EF_AUSS_2_trip_error : BOOL;
	EF_AUSS_2_dcs_occupied : BOOL;

	EF_AUSS_2_status_Filter : ErrorFilter;
	EF_AUSS_2_trip_Filter : ErrorFilter;


(****************************************)


	EF_AUSS_3_status AT%I* : BOOL;
	EF_AUSS_3_trip AT%I* : BOOL;
	EF_AUSS_3_mode AT%I* : BOOL;

	EF_AUSS_3_trigger : BOOL;
	EF_AUSS_3_latch : BOOL;
	EF_AUSS_3_common_alarm : BOOL;
	EF_AUSS_3_status_error : BOOL;
	EF_AUSS_3_trip_error : BOOL;
	EF_AUSS_3_dcs_occupied : BOOL;

	EF_AUSS_3_status_Filter : ErrorFilter;
	EF_AUSS_3_trip_Filter : ErrorFilter;

(*******************************************************)


	FB_EDH_AUSS_3: Flowchart_5_6;
	EDH_AUSS_3_on_status : BOOL;
	EDH_AUSS_3_flow_status AT%I* : BOOL;
	EDH_AUSS_3_high_temp AT%I* : BOOL;

	EDH_AUSS_3_common_alarm : BOOL;
	EDH_AUSS_3_hightemp_error : BOOL;

(*******************************************************)

	MD_AUSS_1_damper_open AT%I* : BOOL;
	MD_AUSS_1_damper_close AT%I* : BOOL;

	MD_AUSS_2_damper_open AT%I* : BOOL;
	MD_AUSS_2_damper_close AT%I* : BOOL;

	MD_AUSS_3_damper_open AT%I* : BOOL;
	MD_AUSS_3_damper_close AT%I* : BOOL;

	MD_EF_AUSS_2_damper_open AT%I* : BOOL;
	MD_EF_AUSS_2_damper_close AT%I* : BOOL;

	MFD_AUSS_1_damper_open AT%I* : BOOL;
	MFD_AUSS_1_damper_close AT%I* : BOOL;

	MFD_AUSS_2_damper_open AT%I* : BOOL;
	MFD_AUSS_2_damper_close AT%I* : BOOL;

	MFD_AUSS_3_damper_open AT%I* : BOOL;
	MFD_AUSS_3_damper_close AT%I* : BOOL;

	MFD_AUSS_4_damper_open AT%I* : BOOL;
	MFD_AUSS_4_damper_close AT%I* : BOOL;

	MFD_AUSS_5_damper_open AT%I* : BOOL;
	MFD_AUSS_5_damper_close AT%I* : BOOL;

	MFD_AUSS_6_damper_open AT%I* : BOOL;
	MFD_AUSS_6_damper_close AT%I* : BOOL;

	MFD_AUSS_7_damper_open AT%I* : BOOL;
	MFD_AUSS_7_damper_close AT%I* : BOOL;

	MFD_AUSS_8_damper_open AT%I* : BOOL;
	MFD_AUSS_8_damper_close AT%I* : BOOL;

	MFD_AUSS_9_damper_open AT%I* : BOOL;
	MFD_AUSS_9_damper_close AT%I* : BOOL;

(*********************************************************************)
	common_alarm AT%Q* : BOOL;
	dcs_occupied AT%Q* : BOOL;


END_VAR
AHU_AUSS_1_status_Filter(IN:=(NOT AHU_AUSS_1_status AND AHU_AUSS_1_latch),Q=>AHU_AUSS_1_status_error);
AHU_AUSS_1_trip_Filter(IN:=(AHU_AUSS_1_trip AND AHU_AUSS_1_latch),Q=>AHU_AUSS_1_trip_error);
AHU_AUSS_1_common_alarm := AHU_AUSS_1_fire OR AHU_AUSS_1_gas OR AHU_AUSS_1_smoke OR AHU_AUSS_1_status_error OR AHU_AUSS_1_trip_error;


AHU_AUSS_2_status_Filter(IN:=(NOT AHU_AUSS_2_status AND AHU_AUSS_2_latch),Q=>AHU_AUSS_2_status_error);
AHU_AUSS_2_trip_Filter(IN:=(AHU_AUSS_2_trip AND AHU_AUSS_2_latch),Q=>AHU_AUSS_2_trip_error);
AHU_AUSS_2_common_alarm := AHU_AUSS_2_fire OR AHU_AUSS_2_gas OR AHU_AUSS_2_smoke OR AHU_AUSS_2_status_error OR AHU_AUSS_2_trip_error;


AHU_AUSS_common_alarm := AHU_AUSS_1_common_alarm OR AHU_AUSS_2_common_alarm;
AHU_AUSS_dcs_occupied := AHU_AUSS_1_dcs_occupied OR AHU_AUSS_2_dcs_occupied;

	FB_AHU_AUSS(
	ON1:=AHU_AUSS_1_trigger ,
	ON2:=AHU_AUSS_2_trigger ,
	ON3:=FALSE ,
	status_error_1:= AHU_AUSS_1_status_error,
	status_error_2:=AHU_AUSS_2_status_error ,
	status_error_3:=FALSE ,
	trip_error_1:=AHU_AUSS_1_trip_error ,
	trip_error_2:=AHU_AUSS_2_trip_error ,
	trip_error_3:=FALSE ,
	Latch1:=AHU_AUSS_1_latch ,
	Latch2:=AHU_AUSS_2_latch ,
	Latch3:=AHU_AUSS_dummy ,
	DcsOccupied_1=>AHU_AUSS_1_dcs_occupied ,
	DcsOccupied_2=>AHU_AUSS_2_dcs_occupied ,
	DcsOccupied_3=> );


(*********************************)

EF_AUSS_1_status_Filter(IN:=(NOT EF_AUSS_1_status AND EF_AUSS_1_latch),Q=>EF_AUSS_1_status_error);
EF_AUSS_1_trip_Filter(IN:=(EF_AUSS_1_trip AND EF_AUSS_1_latch),Q=>EF_AUSS_1_trip_error);
EF_AUSS_1_common_alarm := EF_AUSS_1_status_error OR EF_AUSS_1_trip_error;

EF_AUSS_2_status_Filter(IN:=(NOT EF_AUSS_2_status AND EF_AUSS_2_latch),Q=>EF_AUSS_2_status_error);
EF_AUSS_2_trip_Filter(IN:=(EF_AUSS_2_trip AND EF_AUSS_2_latch),Q=>EF_AUSS_2_trip_error);
EF_AUSS_2_common_alarm := EF_AUSS_2_status_error OR EF_AUSS_2_trip_error;


EF_AUSS_common_alarm := EF_AUSS_1_common_alarm OR EF_AUSS_2_common_alarm;
EF_AUSS_dcs_occupied := EF_AUSS_1_dcs_occupied OR EF_AUSS_2_dcs_occupied;

	FB_EF_AUSS(
	ON1:=EF_AUSS_1_trigger ,
	ON2:=EF_AUSS_2_trigger ,
	ON3:=FALSE ,
	status_error_1:= EF_AUSS_1_status_error,
	status_error_2:=EF_AUSS_2_status_error ,
	status_error_3:=FALSE ,
	trip_error_1:=EF_AUSS_1_trip_error ,
	trip_error_2:=EF_AUSS_2_trip_error ,
	trip_error_3:=FALSE ,
	Latch1:=EF_AUSS_1_latch ,
	Latch2:=EF_AUSS_2_latch ,
	Latch3:=EF_AUSS_dummy ,
	DcsOccupied_1=>EF_AUSS_1_dcs_occupied ,
	DcsOccupied_2=>EF_AUSS_2_dcs_occupied ,
	DcsOccupied_3=> );

(******************************************************)

EF_AUSS_3_latch := TRUE;

EF_AUSS_3_status_Filter(IN:=(NOT EF_AUSS_3_status AND EF_AUSS_3_latch),Q=>EF_AUSS_3_status_error);
EF_AUSS_3_trip_Filter(IN:=(EF_AUSS_3_trip AND EF_AUSS_3_latch),Q=>EF_AUSS_3_trip_error);
EF_AUSS_3_common_alarm := EF_AUSS_3_status_error OR EF_AUSS_3_trip_error;

(******************************************************)

EDH_AUSS_3_on_status := AHU_AUSS_dcs_occupied;

EDH_AUSS_3_hightemp_error := EDH_AUSS_3_high_temp;
EDH_AUSS_3_common_alarm := EDH_AUSS_3_hightemp_error;

FB_EDH_AUSS_3(on_status:= EDH_AUSS_3_on_status , flow_status:= EDH_AUSS_3_flow_status , high_temp:= EDH_AUSS_3_high_temp);

(*****************************************************)

common_alarm := AHU_AUSS_common_alarm OR EF_AUSS_common_alarm OR EF_AUSS_3_common_alarm OR EDH_AUSS_3_common_alarm;
dcs_occupied := AHU_AUSS_dcs_occupied OR EF_AUSS_dcs_occupied;
END_PROGRAM

(* POU Laboratory, ST *)
PROGRAM Laboratory
VAR

	AHU_LAB_common_alarm : BOOL;
	AHU_LAB_dcs_occupied : BOOL;

	FB_AHU_LAB: Flowchart_1_2_CTRL;

	AHU_LAB_1_status AT%I* : BOOL;
	AHU_LAB_1_trip AT%I* : BOOL;
	AHU_LAB_1_mode AT%I* : BOOL;
	AHU_LAB_1_belt AT%I* : BOOL;
	AHU_LAB_1_fire AT%I* : BOOL;
	AHU_LAB_1_gas AT%I* : BOOL;
	AHU_LAB_1_smoke AT%I* : BOOL;

	AHU_LAB_1_trigger : BOOL;
	AHU_LAB_1_latch : BOOL;
	AHU_LAB_1_common_alarm : BOOL;
	AHU_LAB_1_status_error : BOOL;
	AHU_LAB_1_trip_error : BOOL;
	AHU_LAB_1_dcs_occupied : BOOL;

	AHU_LAB_1_status_Filter : ErrorFilter;
	AHU_LAB_1_trip_Filter : ErrorFilter;

	AHU_LAB_2_status AT%I* : BOOL;
	AHU_LAB_2_trip AT%I* : BOOL;
	AHU_LAB_2_mode AT%I* : BOOL;
	AHU_LAB_2_belt AT%I* : BOOL;
	AHU_LAB_2_fire AT%I* : BOOL;
	AHU_LAB_2_gas AT%I* : BOOL;
	AHU_LAB_2_smoke AT%I* : BOOL;

	AHU_LAB_2_trigger : BOOL;
	AHU_LAB_2_latch : BOOL;
	AHU_LAB_2_common_alarm : BOOL;
	AHU_LAB_2_status_error : BOOL;
	AHU_LAB_2_trip_error : BOOL;
	AHU_LAB_2_dcs_occupied : BOOL;

	AHU_LAB_2_status_Filter : ErrorFilter;
	AHU_LAB_2_trip_Filter : ErrorFilter;


	AHU_LAB_3_status AT%I* : BOOL;
	AHU_LAB_3_trip AT%I* : BOOL;
	AHU_LAB_3_mode AT%I* : BOOL;
	AHU_LAB_3_belt AT%I* : BOOL;
	AHU_LAB_3_fire AT%I* : BOOL;
	AHU_LAB_3_gas AT%I* : BOOL;
	AHU_LAB_3_smoke AT%I* : BOOL;

	AHU_LAB_3_trigger : BOOL;
	AHU_LAB_3_latch : BOOL;
	AHU_LAB_3_common_alarm : BOOL;
	AHU_LAB_3_status_error : BOOL;
	AHU_LAB_3_trip_error : BOOL;
	AHU_LAB_3_dcs_occupied : BOOL;

	AHU_LAB_3_status_Filter : ErrorFilter;
	AHU_LAB_3_trip_Filter : ErrorFilter;

(******************************************************************)

	EF_LAB_common_alarm : BOOL;
	EF_LAB_dcs_occupied : BOOL;

	EF_LAB_dummy : BOOL;
	FB_EF_LAB: Flowchart_3_4_CTRL;

	EF_LAB_1_status AT%I* : BOOL;
	EF_LAB_1_trip AT%I* : BOOL;
	EF_LAB_1_mode AT%I* : BOOL;

	EF_LAB_1_trigger : BOOL;
	EF_LAB_1_latch : BOOL;
	EF_LAB_1_common_alarm : BOOL;
	EF_LAB_1_status_error : BOOL;
	EF_LAB_1_trip_error : BOOL;
	EF_LAB_1_dcs_occupied : BOOL;

	EF_LAB_1_status_Filter : ErrorFilter;
	EF_LAB_1_trip_Filter : ErrorFilter;


	EF_LAB_2_status AT%I* : BOOL;
	EF_LAB_2_trip AT%I* : BOOL;
	EF_LAB_2_mode AT%I* : BOOL;

	EF_LAB_2_trigger : BOOL;
	EF_LAB_2_latch : BOOL;
	EF_LAB_2_common_alarm : BOOL;
	EF_LAB_2_status_error : BOOL;
	EF_LAB_2_trip_error : BOOL;
	EF_LAB_2_dcs_occupied : BOOL;

	EF_LAB_2_status_Filter : ErrorFilter;
	EF_LAB_2_trip_Filter : ErrorFilter;

	FB_EF_LAB_3: Flowchart_7;

	EF_LAB_3_status AT%I* : BOOL;
	EF_LAB_3_trip AT%I* : BOOL;
	EF_LAB_3_mode AT%I* : BOOL;

	EF_LAB_3_trigger : BOOL;
	EF_LAB_3_latch : BOOL;
	EF_LAB_3_common_alarm : BOOL;
	EF_LAB_3_status_error : BOOL;
	EF_LAB_3_trip_error : BOOL;
	EF_LAB_3_dcs_occupied : BOOL;

	EF_LAB_3_status_Filter : ErrorFilter;
	EF_LAB_3_trip_Filter : ErrorFilter;




(******************************************************************)

	FB_EH_LAB_1: Flowchart_5_6;

	EH_LAB_1_on_status : BOOL;
	EH_LAB_1_flow_status AT%I* : BOOL;
	EH_LAB_1_high_temp AT%I* : BOOL;

	EH_LAB_1_common_alarm : BOOL;
	EH_LAB_1_hightemp_error : BOOL;

(*****************************************************************)
	MD_LAB_1_damper_open AT%I* : BOOL;
	MD_LAB_1_damper_close AT%I* : BOOL;

	MD_LAB_2_damper_open AT%I* : BOOL;
	MD_LAB_2_damper_close AT%I* : BOOL;

	MD_LAB_3_damper_open AT%I* : BOOL;
	MD_LAB_3_damper_close AT%I* : BOOL;

	MD_LAB_4_damper_open AT%I* : BOOL;
	MD_LAB_4_damper_close AT%I* : BOOL;

(***************************************************************************)

	common_alarm AT%Q* :BOOL;
	dcs_occupied AT%Q* : BOOL;

END_VAR
AHU_LAB_1_status_Filter(IN:=(NOT AHU_LAB_1_status AND AHU_LAB_1_latch),Q=>AHU_LAB_1_status_error);
AHU_LAB_1_trip_Filter(IN:=(AHU_LAB_1_trip AND AHU_LAB_1_latch),Q=>AHU_LAB_1_trip_error);
AHU_LAB_1_common_alarm := AHU_LAB_1_fire OR AHU_LAB_1_gas OR AHU_LAB_1_smoke OR AHU_LAB_1_status_error OR AHU_LAB_1_trip_error;



AHU_LAB_2_status_Filter(IN:=(NOT AHU_LAB_2_status AND AHU_LAB_2_latch),Q=>AHU_LAB_2_status_error);
AHU_LAB_2_trip_Filter(IN:=(AHU_LAB_2_trip AND AHU_LAB_2_latch),Q=>AHU_LAB_2_trip_error);
AHU_LAB_2_common_alarm := AHU_LAB_2_fire OR AHU_LAB_2_gas OR AHU_LAB_2_smoke OR AHU_LAB_2_status_error OR AHU_LAB_2_trip_error;



AHU_LAB_3_status_Filter(IN:=(NOT AHU_LAB_3_status AND AHU_LAB_3_latch),Q=>AHU_LAB_3_status_error);
AHU_LAB_3_trip_Filter(IN:=(AHU_LAB_3_trip AND AHU_LAB_3_latch),Q=>AHU_LAB_3_trip_error);
AHU_LAB_3_common_alarm := AHU_LAB_3_fire OR AHU_LAB_3_gas OR AHU_LAB_3_smoke OR AHU_LAB_3_status_error OR AHU_LAB_3_trip_error;


AHU_LAB_common_alarm := AHU_LAB_1_common_alarm OR AHU_LAB_2_common_alarm OR AHU_LAB_3_common_alarm;
AHU_LAB_dcs_occupied := AHU_LAB_1_dcs_occupied OR AHU_LAB_2_dcs_occupied OR AHU_LAB_3_dcs_occupied;

	FB_AHU_LAB(
	ON1:=AHU_LAB_1_trigger ,
	ON2:=AHU_LAB_2_trigger ,
	ON3:=AHU_LAB_3_trigger ,
	status_error_1:= AHU_LAB_1_status_error,
	status_error_2:=AHU_LAB_2_status_error ,
	status_error_3:=AHU_LAB_3_status_error ,
	trip_error_1:=AHU_LAB_1_trip_error ,
	trip_error_2:=AHU_LAB_2_trip_error ,
	trip_error_3:=AHU_LAB_3_trip_error ,
	Latch1:=AHU_LAB_1_latch ,
	Latch2:=AHU_LAB_2_latch ,
	Latch3:=AHU_LAB_3_latch ,
	DcsOccupied_1=>AHU_LAB_1_dcs_occupied ,
	DcsOccupied_2=>AHU_LAB_2_dcs_occupied ,
	DcsOccupied_3=>AHU_LAB_3_dcs_occupied );


(********************************************************************)

EF_LAB_1_status_Filter(IN:=(NOT EF_LAB_1_status AND EF_LAB_1_latch),Q=>EF_LAB_1_status_error);
EF_LAB_1_trip_Filter(IN:=(EF_LAB_1_trip AND EF_LAB_1_latch),Q=>EF_LAB_1_trip_error);
EF_LAB_1_common_alarm := EF_LAB_1_status_error OR EF_LAB_1_trip_error;


EF_LAB_2_status_Filter(IN:=(NOT EF_LAB_2_status AND EF_LAB_2_latch),Q=>EF_LAB_2_status_error);
EF_LAB_2_trip_Filter(IN:=(EF_LAB_2_trip AND EF_LAB_2_latch),Q=>EF_LAB_2_trip_error);
EF_LAB_2_common_alarm := EF_LAB_2_status_error OR EF_LAB_2_trip_error;



	FB_EF_LAB(
	ON1:=EF_LAB_1_trigger ,
	ON2:=EF_LAB_2_trigger ,
	ON3:=FALSE ,
	status_error_1:= EF_LAB_1_status_error,
	status_error_2:=EF_LAB_2_status_error ,
	status_error_3:=FALSE ,
	trip_error_1:=EF_LAB_1_trip_error ,
	trip_error_2:=EF_LAB_2_trip_error ,
	trip_error_3:=FALSE ,
	Latch1:=EF_LAB_1_latch ,
	Latch2:=EF_LAB_2_latch ,
	Latch3:=EF_LAB_dummy ,
	DcsOccupied_1=>EF_LAB_1_dcs_occupied ,
	DcsOccupied_2=>EF_LAB_2_dcs_occupied ,
	DcsOccupied_3=> );




EF_LAB_3_status_Filter(IN:=(NOT EF_LAB_3_status AND EF_LAB_3_latch),Q=>EF_LAB_3_status_error);
EF_LAB_3_trip_Filter(IN:=(EF_LAB_3_trip AND EF_LAB_3_latch),Q=>EF_LAB_3_trip_error);
EF_LAB_3_common_alarm := EF_LAB_3_status_error OR EF_LAB_3_trip_error;



FB_EF_LAB_3(
Trigger:=EF_LAB_3_trigger ,
Latch:=EF_LAB_3_latch ,
DCS_Occupied=>EF_LAB_3_dcs_occupied );


EF_LAB_common_alarm := EF_LAB_1_common_alarm OR EF_LAB_2_common_alarm OR EF_LAB_3_dcs_occupied ;
EF_LAB_dcs_occupied := EF_LAB_1_dcs_occupied OR EF_LAB_2_dcs_occupied OR EF_LAB_3_dcs_occupied;


(*******************************************************************)

EH_LAB_1_on_status := AHU_LAB_dcs_occupied;
EH_LAB_1_hightemp_error := EH_LAB_1_high_temp;
EH_LAB_1_common_alarm := EH_LAB_1_hightemp_error;

FB_EH_LAB_1(on_status:= EH_LAB_1_on_status , flow_status:= EH_LAB_1_flow_status , high_temp:= EH_LAB_1_high_temp);

(*******************************************************************)

common_alarm := AHU_LAB_dcs_occupied OR EF_LAB_common_alarm OR EH_LAB_1_common_alarm;
dcs_occupied := AHU_LAB_dcs_occupied OR EF_LAB_dcs_occupied;
END_PROGRAM

(* POU MainSwitchBoard, ST *)
PROGRAM MainSwitchBoard
VAR

	AHU_MSB_common_alarm : BOOL;
	AHU_MSB_dcs_occupied : BOOL;

	FB_AHU_MSB: Flowchart_1_2_CTRL;

	AHU_MSB_1A_status AT%I* : BOOL;
	AHU_MSB_1A_trip AT%I* : BOOL;
	AHU_MSB_1A_mode AT%I* : BOOL;
	AHU_MSB_1A_belt AT%I* : BOOL;
	AHU_MSB_1A_fire AT%I* : BOOL;
	AHU_MSB_1A_gas AT%I* : BOOL;
	AHU_MSB_1A_smoke AT%I* : BOOL;

	AHU_MSB_1A_trigger : BOOL;
	AHU_MSB_1A_latch : BOOL;
	AHU_MSB_1A_common_alarm : BOOL;
	AHU_MSB_1A_status_error : BOOL;
	AHU_MSB_1A_trip_error : BOOL;
	AHU_MSB_1A_dcs_occupied : BOOL;

	AHU_MSB_1A_status_Filter : ErrorFilter;
	AHU_MSB_1A_trip_Filter : ErrorFilter;


	AHU_MSB_1B_status AT%I* : BOOL;
	AHU_MSB_1B_trip AT%I* : BOOL;
	AHU_MSB_1B_mode AT%I* : BOOL;
	AHU_MSB_1B_belt AT%I* : BOOL;
	AHU_MSB_1B_fire AT%I* : BOOL;
	AHU_MSB_1B_gas AT%I* : BOOL;
	AHU_MSB_1B_smoke AT%I* : BOOL;

	AHU_MSB_1B_trigger : BOOL;
	AHU_MSB_1B_latch : BOOL;
	AHU_MSB_1B_common_alarm : BOOL;
	AHU_MSB_1B_status_error : BOOL;
	AHU_MSB_1B_trip_error : BOOL;
	AHU_MSB_1B_dcs_occupied : BOOL;

	AHU_MSB_1B_status_Filter : ErrorFilter;
	AHU_MSB_1B_trip_Filter : ErrorFilter;



	AHU_MSB_1C_status AT%I* : BOOL;
	AHU_MSB_1C_trip AT%I* : BOOL;
	AHU_MSB_1C_mode AT%I* : BOOL;
	AHU_MSB_1C_belt AT%I* : BOOL;
	AHU_MSB_1C_fire AT%I* : BOOL;
	AHU_MSB_1C_gas AT%I* : BOOL;
	AHU_MSB_1C_smoke AT%I* : BOOL;

	AHU_MSB_1C_trigger : BOOL;
	AHU_MSB_1C_latch : BOOL;
	AHU_MSB_1C_common_alarm : BOOL;
	AHU_MSB_1C_status_error : BOOL;
	AHU_MSB_1C_trip_error : BOOL;
	AHU_MSB_1C_dcs_occupied : BOOL;

	AHU_MSB_1C_status_Filter : ErrorFilter;
	AHU_MSB_1C_trip_Filter : ErrorFilter;

(***************************************************************)


	EF_MSB_common_alarm : BOOL;
	EF_MSB_dcs_occupied : BOOL;

	EF_MSB_dummy : BOOL;
	FB_EF_MSB: Flowchart_3_4_CTRL;

	EF_MSB_1_status AT%I* : BOOL;
	EF_MSB_1_trip AT%I* : BOOL;
	EF_MSB_1_mode AT%I* : BOOL;

	EF_MSB_1_trigger : BOOL;
	EF_MSB_1_latch : BOOL;
	EF_MSB_1_common_alarm : BOOL;
	EF_MSB_1_status_error : BOOL;
	EF_MSB_1_trip_error : BOOL;
	EF_MSB_1_dcs_occupied : BOOL;

	EF_MSB_1_status_Filter : ErrorFilter;
	EF_MSB_1_trip_Filter : ErrorFilter;


	EF_MSB_2_status AT%I* : BOOL;
	EF_MSB_2_trip AT%I* : BOOL;
	EF_MSB_2_mode AT%I* : BOOL;

	EF_MSB_2_trigger : BOOL;
	EF_MSB_2_latch : BOOL;
	EF_MSB_2_common_alarm : BOOL;
	EF_MSB_2_status_error : BOOL;
	EF_MSB_2_trip_error : BOOL;
	EF_MSB_2_dcs_occupied : BOOL;

	EF_MSB_2_status_Filter : ErrorFilter;
	EF_MSB_2_trip_Filter : ErrorFilter;


	EF_MSB_common_alarm_2 : BOOL;
	EF_MSB_dcs_occupied_2 : BOOL;

	EF_MSB_dummy_2 : BOOL;
	FB_EF_MSB_2: Flowchart_3_4_CTRL;

	EF_MSB_3_status AT%I* : BOOL;
	EF_MSB_3_trip AT%I* : BOOL;
	EF_MSB_3_mode AT%I* : BOOL;

	EF_MSB_3_trigger : BOOL;
	EF_MSB_3_latch : BOOL;
	EF_MSB_3_common_alarm : BOOL;
	EF_MSB_3_status_error : BOOL;
	EF_MSB_3_trip_error : BOOL;
	EF_MSB_3_dcs_occupied : BOOL;

	EF_MSB_3_status_Filter : ErrorFilter;
	EF_MSB_3_trip_Filter : ErrorFilter;



	EF_MSB_4_status AT%I* : BOOL;
	EF_MSB_4_trip AT%I* : BOOL;
	EF_MSB_4_mode AT%I* : BOOL;

	EF_MSB_4_trigger : BOOL;
	EF_MSB_4_latch : BOOL;
	EF_MSB_4_common_alarm : BOOL;
	EF_MSB_4_status_error : BOOL;
	EF_MSB_4_trip_error : BOOL;
	EF_MSB_4_dcs_occupied : BOOL;

	EF_MSB_4_status_Filter : ErrorFilter;
	EF_MSB_4_trip_Filter : ErrorFilter;

(***************************************************************)

	FB_EDH_MSB_1: Flowchart_5_6;

	EDH_MSB_1_on_status AT%I* : BOOL;
	EDH_MSB_1_flow_status AT%I* : BOOL;
	EDH_MSB_1_high_temp AT%I* : BOOL;

	EDH_MSB_1_common_alarm : BOOL;
	EDH_MSB_1_hightemp_error : BOOL;

(***************************************************************)

	MD_MSB_01A_damper_open AT%I* : BOOL;
	MD_MSB_01A_damper_close AT%I* : BOOL;

	MD_MSB_01B_damper_open AT%I* : BOOL;
	MD_MSB_01B_damper_close AT%I* : BOOL;

	MD_MSB_01C_damper_open AT%I* : BOOL;
	MD_MSB_01C_damper_close AT%I* : BOOL;

	MD_MSB_01D_damper_open AT%I* : BOOL;
	MD_MSB_01D_damper_close AT%I* : BOOL;

(***************************************************************)

	MD_EF_MSB_01E_damper_open AT%I* : BOOL;
	MD_EF_MSB_01E_damper_close AT%I* : BOOL;

	MD_EF_MSB_01F_damper_open AT%I* : BOOL;
	MD_EF_MSB_01F_damper_close AT%I* : BOOL;

(***************************************************************)

	MFD_MSB_1_damper_open AT%I* : BOOL;
	MFD_MSB_1_damper_close AT%I* : BOOL;

	MFD_MSB_2_damper_open AT%I* : BOOL;
	MFD_MSB_2_damper_close AT%I* : BOOL;

	MFD_MSB_3_damper_open AT%I* : BOOL;
	MFD_MSB_3_damper_close AT%I* : BOOL;

	MFD_MSB_4_damper_open AT%I* : BOOL;
	MFD_MSB_4_damper_close AT%I* : BOOL;

	MFD_MSB_5_damper_open AT%I* : BOOL;
	MFD_MSB_5_damper_close AT%I* : BOOL;

	MFD_MSB_6_damper_open AT%I* : BOOL;
	MFD_MSB_6_damper_close AT%I* : BOOL;

	MFD_MSB_7_damper_open AT%I* : BOOL;
	MFD_MSB_7_damper_close AT%I* : BOOL;

	MFD_MSB_8_damper_open AT%I* : BOOL;
	MFD_MSB_8_damper_close AT%I* : BOOL;

	MFD_MSB_9_damper_open AT%I* : BOOL;
	MFD_MSB_9_damper_close AT%I* : BOOL;
(*******************************************************************)
	common_alarm AT%Q* : BOOL;
	dcs_occupied AT%Q* : BOOL;

END_VAR
AHU_MSB_1A_status_Filter(IN:=(NOT AHU_MSB_1A_status AND AHU_MSB_1A_latch),Q=>AHU_MSB_1A_status_error);
AHU_MSB_1A_trip_Filter(IN:=(AHU_MSB_1A_trip AND AHU_MSB_1A_latch),Q=>AHU_MSB_1A_trip_error);
AHU_MSB_1A_common_alarm := AHU_MSB_1A_fire OR AHU_MSB_1A_gas OR AHU_MSB_1A_smoke OR AHU_MSB_1A_status_error OR AHU_MSB_1A_trip_error;


AHU_MSB_1B_status_Filter(IN:=(NOT AHU_MSB_1B_status AND AHU_MSB_1B_latch),Q=>AHU_MSB_1B_status_error);
AHU_MSB_1B_trip_Filter(IN:=(AHU_MSB_1B_trip AND AHU_MSB_1B_latch),Q=>AHU_MSB_1B_trip_error);
AHU_MSB_1B_common_alarm := AHU_MSB_1B_fire OR AHU_MSB_1B_gas OR AHU_MSB_1B_smoke OR AHU_MSB_1B_status_error OR AHU_MSB_1B_trip_error;


AHU_MSB_1C_status_Filter(IN:=(NOT AHU_MSB_1C_status AND AHU_MSB_1C_latch),Q=>AHU_MSB_1C_status_error);
AHU_MSB_1C_trip_Filter(IN:=(AHU_MSB_1C_trip AND AHU_MSB_1C_latch),Q=>AHU_MSB_1C_trip_error);
AHU_MSB_1C_common_alarm := AHU_MSB_1C_fire OR AHU_MSB_1C_gas OR AHU_MSB_1C_smoke OR AHU_MSB_1C_status_error OR AHU_MSB_1C_trip_error;


AHU_MSB_common_alarm := AHU_MSB_1A_common_alarm OR AHU_MSB_1B_common_alarm OR AHU_MSB_1C_common_alarm;
AHU_MSB_dcs_occupied := AHU_MSB_1A_dcs_occupied OR AHU_MSB_1B_dcs_occupied OR AHU_MSB_1C_dcs_occupied;

	FB_AHU_MSB(
	ON1:=AHU_MSB_1A_trigger ,
	ON2:=AHU_MSB_1B_trigger ,
	ON3:=AHU_MSB_1C_trigger ,
	status_error_1:= AHU_MSB_1A_status_error,
	status_error_2:=AHU_MSB_1B_status_error ,
	status_error_3:=AHU_MSB_1C_status_error ,
	trip_error_1:=AHU_MSB_1A_trip_error ,
	trip_error_2:=AHU_MSB_1B_trip_error ,
	trip_error_3:=AHU_MSB_1C_trip_error ,
	Latch1:=AHU_MSB_1A_latch ,
	Latch2:=AHU_MSB_1B_latch ,
	Latch3:=AHU_MSB_1C_latch ,
	DcsOccupied_1=>AHU_MSB_1A_dcs_occupied ,
	DcsOccupied_2=>AHU_MSB_1B_dcs_occupied ,
	DcsOccupied_3=>AHU_MSB_1C_dcs_occupied );

(***************************************************************)


EF_MSB_1_status_Filter(IN:=(NOT EF_MSB_1_status AND EF_MSB_1_latch),Q=>EF_MSB_1_status_error);
EF_MSB_1_trip_Filter(IN:=(EF_MSB_1_trip AND EF_MSB_1_latch),Q=>EF_MSB_1_trip_error);
EF_MSB_1_common_alarm := EF_MSB_1_status_error OR EF_MSB_1_trip_error;


EF_MSB_2_status_Filter(IN:=(NOT EF_MSB_2_status AND EF_MSB_2_latch),Q=>EF_MSB_2_status_error);
EF_MSB_2_trip_Filter(IN:=(EF_MSB_2_trip AND EF_MSB_2_latch),Q=>EF_MSB_2_trip_error);
EF_MSB_2_common_alarm := EF_MSB_2_status_error OR EF_MSB_2_trip_error;


EF_MSB_common_alarm := EF_MSB_1_common_alarm OR EF_MSB_2_common_alarm;
EF_MSB_dcs_occupied := EF_MSB_1_dcs_occupied OR EF_MSB_2_dcs_occupied;

	FB_EF_MSB(
	ON1:=EF_MSB_1_trigger ,
	ON2:=EF_MSB_2_trigger ,
	ON3:=FALSE ,
	status_error_1:= EF_MSB_1_status_error,
	status_error_2:=EF_MSB_2_status_error ,
	status_error_3:=FALSE ,
	trip_error_1:=EF_MSB_1_trip_error ,
	trip_error_2:=EF_MSB_2_trip_error ,
	trip_error_3:=FALSE ,
	Latch1:=EF_MSB_1_latch ,
	Latch2:=EF_MSB_2_latch ,
	Latch3:=EF_MSB_dummy ,
	DcsOccupied_1=>EF_MSB_1_dcs_occupied ,
	DcsOccupied_2=>EF_MSB_2_dcs_occupied ,
	DcsOccupied_3=> );

EF_MSB_3_status_Filter(IN:=(NOT EF_MSB_3_status AND EF_MSB_3_latch),Q=>EF_MSB_3_status_error);
EF_MSB_3_trip_Filter(IN:=(EF_MSB_3_trip AND EF_MSB_3_latch),Q=>EF_MSB_3_trip_error);
EF_MSB_3_common_alarm := EF_MSB_3_status_error OR EF_MSB_3_trip_error;


EF_MSB_4_status_Filter(IN:=(NOT EF_MSB_4_status AND EF_MSB_4_latch),Q=>EF_MSB_4_status_error);
EF_MSB_4_trip_Filter(IN:=(EF_MSB_4_trip AND EF_MSB_4_latch),Q=>EF_MSB_4_trip_error);
EF_MSB_4_common_alarm := EF_MSB_4_status_error OR EF_MSB_4_trip_error;

EF_MSB_common_alarm_2 := EF_MSB_3_common_alarm OR EF_MSB_4_common_alarm;
EF_MSB_dcs_occupied_2 := EF_MSB_3_dcs_occupied OR EF_MSB_4_dcs_occupied;

	FB_EF_MSB_2(
	ON1:=EF_MSB_3_trigger ,
	ON2:=EF_MSB_4_trigger ,
	ON3:=FALSE ,
	status_error_1:= EF_MSB_3_status_error,
	status_error_2:=EF_MSB_4_status_error ,
	status_error_3:=FALSE ,
	trip_error_1:=EF_MSB_3_trip_error ,
	trip_error_2:=EF_MSB_4_trip_error ,
	trip_error_3:=FALSE ,
	Latch1:=EF_MSB_3_latch ,
	Latch2:=EF_MSB_4_latch ,
	Latch3:=EF_MSB_dummy ,
	DcsOccupied_1=>EF_MSB_3_dcs_occupied ,
	DcsOccupied_2=>EF_MSB_4_dcs_occupied ,
	DcsOccupied_3=> );

(***************************************************************)

EDH_MSB_1_on_status := AHU_MSB_dcs_occupied;
EDH_MSB_1_hightemp_error := EDH_MSB_1_high_temp;
EDH_MSB_1_common_alarm := EDH_MSB_1_hightemp_error;

FB_EDH_MSB_1(on_status:= EDH_MSB_1_on_status , flow_status:= EDH_MSB_1_flow_status , high_temp:= EDH_MSB_1_high_temp);


(***************************************************************)

common_alarm := AHU_MSB_common_alarm OR EF_MSB_common_alarm OR EF_MSB_common_alarm_2;
dcs_occupied := AHU_MSB_dcs_occupied OR EF_MSB_dcs_occupied OR EF_MSB_dcs_occupied_2;
END_PROGRAM

(* POU EDG_HOUSE, ST *)
PROGRAM EDG_HOUSE
VAR

	AHU_EDG_common_alarm : BOOL;
	AHU_EDG_dcs_occupied  : BOOL;

	AHU_EDG_dummy : BOOL;

	FB_AHU_EDG: Flowchart_3_4_CTRL;

	AHU_EDG_1_status AT%I* : BOOL;
	AHU_EDG_1_trip AT%I* : BOOL;
	AHU_EDG_1_mode AT%I* : BOOL;
	AHU_EDG_1_belt AT%I* : BOOL;
	AHU_EDG_1_fire AT%I* : BOOL;
	AHU_EDG_1_gas AT%I* : BOOL;
	AHU_EDG_1_smoke AT%I* : BOOL;

	AHU_EDG_1_trigger : BOOL;
	AHU_EDG_1_latch : BOOL;
	AHU_EDG_1_common_alarm : BOOL;
	AHU_EDG_1_status_error : BOOL;
	AHU_EDG_1_trip_error : BOOL;
	AHU_EDG_1_dcs_occupied : BOOL;

	AHU_EDG_1_status_Filter : ErrorFilter;
	AHU_EDG_1_trip_Filter : ErrorFilter;


	AHU_EDG_2_status AT%I* : BOOL;
	AHU_EDG_2_trip AT%I* : BOOL;
	AHU_EDG_2_mode AT%I* : BOOL;
	AHU_EDG_2_belt AT%I* : BOOL;
	AHU_EDG_2_fire AT%I* : BOOL;
	AHU_EDG_2_gas AT%I* : BOOL;
	AHU_EDG_2_smoke AT%I* : BOOL;

	AHU_EDG_2_trigger : BOOL;
	AHU_EDG_2_latch : BOOL;
	AHU_EDG_2_common_alarm : BOOL;
	AHU_EDG_2_status_error : BOOL;
	AHU_EDG_2_trip_error : BOOL;
	AHU_EDG_2_dcs_occupied : BOOL;

	AHU_EDG_2_status_Filter : ErrorFilter;
	AHU_EDG_2_trip_Filter : ErrorFilter;



(**********************************************************************************************)


	EF_EDG_common_alarm : BOOL;
	EF_EDG_dcs_occupied  : BOOL;

	EF_EDG_dummy : BOOL;

	FB_EF_EDG: Flowchart_3_4_CTRL;

	EF_EDG_1A_status AT%I* : BOOL;
	EF_EDG_1A_trip AT%I* : BOOL;
	EF_EDG_1A_mode AT%I* : BOOL;

	EF_EDG_1A_trigger : BOOL;
	EF_EDG_1A_latch : BOOL;
	EF_EDG_1A_common_alarm : BOOL;
	EF_EDG_1A_status_error : BOOL;
	EF_EDG_1A_trip_error : BOOL;
	EF_EDG_1A_dcs_occupied : BOOL;

	EF_EDG_1A_status_Filter : ErrorFilter;
	EF_EDG_1A_trip_Filter : ErrorFilter;


	EF_EDG_1B_status AT%I* : BOOL;
	EF_EDG_1B_trip AT%I* : BOOL;
	EF_EDG_1B_mode AT%I* : BOOL;

	EF_EDG_1B_trigger : BOOL;
	EF_EDG_1B_latch : BOOL;
	EF_EDG_1B_common_alarm : BOOL;
	EF_EDG_1B_status_error : BOOL;
	EF_EDG_1B_trip_error : BOOL;
	EF_EDG_1B_dcs_occupied : BOOL;

	EF_EDG_1B_status_Filter : ErrorFilter;
	EF_EDG_1B_trip_Filter : ErrorFilter;

(**********************************************************************************************)

	EF_EDG_2_status AT%I* : BOOL;
	EF_EDG_2_trip AT%I* : BOOL;
	EF_EDG_2_mode AT%I* : BOOL;

	EF_EDG_2_trigger : BOOL;
	EF_EDG_2_latch : BOOL;
	EF_EDG_2_common_alarm : BOOL;
	EF_EDG_2_status_error : BOOL;
	EF_EDG_2_trip_error : BOOL;
	EF_EDG_2_dcs_occupied : BOOL;

	EF_EDG_2_status_Filter : ErrorFilter;
	EF_EDG_2_trip_Filter : ErrorFilter;

(**********************************************************************************************)

	MD_EDG_1A_damper_open AT%I* : BOOL;
	MD_EDG_1A_damper_close AT%I* : BOOL;

	MD_EDG_1B_damper_open AT%I* : BOOL;
	MD_EDG_1B_damper_close AT%I* : BOOL;

	MD_EF_EDG_2_damper_open AT%I* : BOOL;
	MD_EF_EDG_2_damper_close AT%I* : BOOL;

(*********************************************************************************************)

	MFD_EDG_1_damper_open AT%I* : BOOL;
	MFD_EDG_1_damper_close AT%I* : BOOL;

	MFD_EDG_2_damper_open AT%I* : BOOL;
	MFD_EDG_2_damper_close AT%I* : BOOL;

	MFD_EDG_3_damper_open AT%I* : BOOL;
	MFD_EDG_3_damper_close AT%I* : BOOL;


(************************************************************************)

	common_alarm AT%Q* : BOOL;
	dcs_occupied AT%Q* : BOOL;


END_VAR
AHU_EDG_1_status_Filter(IN:=(NOT AHU_EDG_1_status AND AHU_EDG_1_latch),Q=>AHU_EDG_1_status_error);
AHU_EDG_1_trip_Filter(IN:=(AHU_EDG_1_trip AND AHU_EDG_1_latch),Q=>AHU_EDG_1_trip_error);
AHU_EDG_1_common_alarm := AHU_EDG_1_fire OR AHU_EDG_1_gas OR AHU_EDG_1_smoke OR AHU_EDG_1_status_error OR AHU_EDG_1_trip_error;

AHU_EDG_2_status_Filter(IN:=(NOT AHU_EDG_2_status AND AHU_EDG_2_latch),Q=>AHU_EDG_2_status_error);
AHU_EDG_2_trip_Filter(IN:=(AHU_EDG_2_trip AND AHU_EDG_2_latch),Q=>AHU_EDG_2_trip_error);
AHU_EDG_2_common_alarm := AHU_EDG_2_fire OR AHU_EDG_2_gas OR AHU_EDG_2_smoke OR AHU_EDG_2_status_error OR AHU_EDG_2_trip_error;


AHU_EDG_common_alarm := AHU_EDG_1_common_alarm OR AHU_EDG_2_common_alarm;
AHU_EDG_dcs_occupied := AHU_EDG_1_dcs_occupied OR AHU_EDG_2_dcs_occupied;

	FB_AHU_EDG(
	ON1:=AHU_EDG_1_trigger ,
	ON2:=AHU_EDG_2_trigger ,
	ON3:=FALSE ,
	status_error_1:= AHU_EDG_1_status_error,
	status_error_2:=AHU_EDG_2_status_error ,
	status_error_3:=FALSE ,
	trip_error_1:=AHU_EDG_1_trip_error ,
	trip_error_2:=AHU_EDG_2_trip_error ,
	trip_error_3:=FALSE ,
	Latch1:=AHU_EDG_1_latch ,
	Latch2:=AHU_EDG_2_latch ,
	Latch3:=AHU_EDG_dummy ,
	DcsOccupied_1=>AHU_EDG_1_dcs_occupied ,
	DcsOccupied_2=>AHU_EDG_2_dcs_occupied ,
	DcsOccupied_3=> );



(**********************************************************************************************)


EF_EDG_1A_status_Filter(IN:=(NOT EF_EDG_1A_status AND EF_EDG_1A_latch),Q=>EF_EDG_1A_status_error);
EF_EDG_1A_trip_Filter(IN:=(EF_EDG_1A_trip AND EF_EDG_1A_latch),Q=>EF_EDG_1A_trip_error);
EF_EDG_1A_common_alarm := EF_EDG_1A_status_error OR EF_EDG_1A_trip_error;

EF_EDG_1B_status_Filter(IN:=(NOT EF_EDG_1B_status AND EF_EDG_1B_latch),Q=>EF_EDG_1B_status_error);
EF_EDG_1B_trip_Filter(IN:=(EF_EDG_1B_trip AND EF_EDG_1B_latch),Q=>EF_EDG_1B_trip_error);
EF_EDG_1B_common_alarm := EF_EDG_1B_status_error OR EF_EDG_1B_trip_error;



EF_EDG_common_alarm := EF_EDG_1A_common_alarm OR EF_EDG_1B_common_alarm;
EF_EDG_dcs_occupied := EF_EDG_1A_dcs_occupied OR EF_EDG_1B_dcs_occupied;

	FB_EF_EDG(
	ON1:=EF_EDG_1A_trigger ,
	ON2:=EF_EDG_1B_trigger ,
	ON3:=FALSE ,
	status_error_1:= EF_EDG_1A_status_error,
	status_error_2:=EF_EDG_1B_status_error ,
	status_error_3:=FALSE ,
	trip_error_1:=EF_EDG_1A_trip_error ,
	trip_error_2:=EF_EDG_1B_trip_error ,
	trip_error_3:=FALSE ,
	Latch1:=EF_EDG_1A_latch ,
	Latch2:=EF_EDG_1B_latch ,
	Latch3:=EF_EDG_dummy ,
	DcsOccupied_1=>EF_EDG_1A_dcs_occupied ,
	DcsOccupied_2=>EF_EDG_1B_dcs_occupied ,
	DcsOccupied_3=> );

(**********************************************************************************************)

EF_EDG_2_latch := TRUE;

EF_EDG_2_status_Filter(IN:=(NOT EF_EDG_2_status AND EF_EDG_2_latch),Q=>EF_EDG_2_status_error);
EF_EDG_2_trip_Filter(IN:=(EF_EDG_2_trip AND EF_EDG_2_latch),Q=>EF_EDG_2_trip_error);
EF_EDG_2_common_alarm := EF_EDG_2_status_error OR EF_EDG_2_trip_error;

(**********************************************************************************************)


common_alarm := AHU_EDG_common_alarm OR AHU_EDG_dcs_occupied;
dcs_occupied := AHU_EDG_dcs_occupied OR EF_EDG_dcs_occupied;
END_PROGRAM

(* POU FieldAuxiliarryRoom2, ST *)
PROGRAM FieldAuxiliarryRoom2
VAR

	AHU_FAR2_common_alarm : BOOL;
	AHU_FAR2_dcs_occupied : BOOL;

	AHU_FAR2_dummy : BOOL;
	FB_AHU_FAR2: Flowchart_3_4_CTRL;

	AHU_FAR2_1_status AT%I* : BOOL;
	AHU_FAR2_1_trip AT%I* : BOOL;
	AHU_FAR2_1_mode AT%I* : BOOL;
	AHU_FAR2_1_belt AT%I* : BOOL;
	AHU_FAR2_1_fire AT%I* : BOOL;
	AHU_FAR2_1_gas AT%I* : BOOL;
	AHU_FAR2_1_smoke AT%I* : BOOL;

	AHU_FAR2_1_trigger : BOOL;
	AHU_FAR2_1_latch : BOOL;
	AHU_FAR2_1_common_alarm : BOOL;
	AHU_FAR2_1_status_error : BOOL;
	AHU_FAR2_1_trip_error : BOOL;
	AHU_FAR2_1_dcs_occupied : BOOL;

	AHU_FAR2_1_status_Filter : ErrorFilter;
	AHU_FAR2_1_trip_Filter : ErrorFilter;




	AHU_FAR2_2_status AT%I* : BOOL;
	AHU_FAR2_2_trip AT%I* : BOOL;
	AHU_FAR2_2_mode AT%I* : BOOL;
	AHU_FAR2_2_belt AT%I* : BOOL;
	AHU_FAR2_2_fire AT%I* : BOOL;
	AHU_FAR2_2_gas AT%I* : BOOL;
	AHU_FAR2_2_smoke AT%I* : BOOL;

	AHU_FAR2_2_trigger : BOOL;
	AHU_FAR2_2_latch : BOOL;
	AHU_FAR2_2_common_alarm : BOOL;
	AHU_FAR2_2_status_error : BOOL;
	AHU_FAR2_2_trip_error : BOOL;
	AHU_FAR2_2_dcs_occupied : BOOL;

	AHU_FAR2_2_status_Filter : ErrorFilter;
	AHU_FAR2_2_trip_Filter : ErrorFilter;

(***)


	EF_FAR2_common_alarm : BOOL;
	EF_FAR2_dcs_occupied : BOOL;

	EF_FAR2_dummy : BOOL;
	FB_EF_FAR2: Flowchart_3_4_CTRL;

	EF_FAR2_1A_status AT%I* : BOOL;
	EF_FAR2_1A_trip AT%I* : BOOL;
	EF_FAR2_1A_mode AT%I* : BOOL;

	EF_FAR2_1A_trigger : BOOL;
	EF_FAR2_1A_latch : BOOL;
	EF_FAR2_1A_common_alarm : BOOL;
	EF_FAR2_1A_status_error : BOOL;
	EF_FAR2_1A_trip_error : BOOL;
	EF_FAR2_1A_dcs_occupied : BOOL;

	EF_FAR2_1A_status_Filter : ErrorFilter;
	EF_FAR2_1A_trip_Filter : ErrorFilter;


	EF_FAR2_1B_status AT%I* : BOOL;
	EF_FAR2_1B_trip AT%I* : BOOL;
	EF_FAR2_1B_mode AT%I* : BOOL;

	EF_FAR2_1B_trigger : BOOL;
	EF_FAR2_1B_latch : BOOL;
	EF_FAR2_1B_common_alarm : BOOL;
	EF_FAR2_1B_status_error : BOOL;
	EF_FAR2_1B_trip_error : BOOL;
	EF_FAR2_1B_dcs_occupied : BOOL;

	EF_FAR2_1B_status_Filter : ErrorFilter;
	EF_FAR2_1B_trip_Filter : ErrorFilter;


(*********************)


	FB_EF_FAR2_3: Flowchart_7;

	EF_FAR2_3_status AT%I* : BOOL;
	EF_FAR2_3_trip AT%I* : BOOL;
	EF_FAR2_3_mode AT%I* : BOOL;

	EF_FAR2_3_trigger : BOOL;
	EF_FAR2_3_latch : BOOL;
	EF_FAR2_3_common_alarm : BOOL;
	EF_FAR2_3_status_error : BOOL;
	EF_FAR2_3_trip_error : BOOL;
	EF_FAR2_3_dcs_occupied : BOOL;

	EF_FAR2_3_status_Filter : ErrorFilter;
	EF_FAR2_3_trip_Filter : ErrorFilter;

(************************************)



	EF_FAR2_2_status AT%I* : BOOL;
	EF_FAR2_2_trip AT%I* : BOOL;
	EF_FAR2_2_mode AT%I* : BOOL;

	EF_FAR2_2_trigger : BOOL;
	EF_FAR2_2_latch : BOOL;
	EF_FAR2_2_common_alarm : BOOL;
	EF_FAR2_2_status_error : BOOL;
	EF_FAR2_2_trip_error : BOOL;
	EF_FAR2_2_dcs_occupied : BOOL;

	EF_FAR2_2_status_Filter : ErrorFilter;
	EF_FAR2_2_trip_Filter : ErrorFilter;

(*************************)

	FB_EDH_FAR2_1: Flowchart_5_6;
	EDH_FAR2_1_on_status : BOOL;
	EDH_FAR2_1_flow_status AT%I* : BOOL;
	EDH_FAR2_1_high_temp AT%I* : BOOL;

	EDH_FAR2_1_common_alarm : BOOL;
	EDH_FAR2_1_hightemp_error : BOOL;




(***************************)

	MD_FAR2_1A_damper_open AT%I* : BOOL;
	MD_FAR2_1A_damper_close AT%I* : BOOL;

	MD_FAR2_1B_damper_open AT%I* : BOOL;
	MD_FAR2_1B_damper_close AT%I* : BOOL;

	MD_FAR2_1C_damper_open AT%I* : BOOL;
	MD_FAR2_1C_damper_close AT%I* : BOOL;

	MD_EF_FAR2_2_damper_open AT%I* : BOOL;
	MD_EF_FAR2_2_damper_close AT%I* : BOOL;

(*************************)

	MFD_FAR2_1_damper_open AT%I* : BOOL;
	MFD_FAR2_1_damper_close AT%I* : BOOL;

	MFD_FAR2_2_damper_open AT%I* : BOOL;
	MFD_FAR2_2_damper_close AT%I* : BOOL;

	MFD_FAR2_3_damper_open AT%I* : BOOL;
	MFD_FAR2_3_damper_close AT%I* : BOOL;

	MFD_FAR2_4_damper_open AT%I* : BOOL;
	MFD_FAR2_4_damper_close AT%I* : BOOL;

	MFD_FAR2_5_damper_open AT%I* : BOOL;
	MFD_FAR2_5_damper_close AT%I* : BOOL;

	MFD_FAR2_6_damper_open AT%I* : BOOL;
	MFD_FAR2_6_damper_close AT%I* : BOOL;

(********************************)
	common_alarm AT%Q* : BOOL;
	dcs_occupied AT%Q* : BOOL;

END_VAR
AHU_FAR2_1_status_Filter(IN:=(NOT AHU_FAR2_1_status AND AHU_FAR2_1_latch),Q=>AHU_FAR2_1_status_error);
AHU_FAR2_1_trip_Filter(IN:=(AHU_FAR2_1_trip AND AHU_FAR2_1_latch),Q=>AHU_FAR2_1_trip_error);
AHU_FAR2_1_common_alarm := AHU_FAR2_1_fire OR AHU_FAR2_1_gas OR AHU_FAR2_1_smoke OR AHU_FAR2_1_status_error OR AHU_FAR2_1_trip_error;


AHU_FAR2_2_status_Filter(IN:=(NOT AHU_FAR2_2_status AND AHU_FAR2_2_latch),Q=>AHU_FAR2_2_status_error);
AHU_FAR2_2_trip_Filter(IN:=(AHU_FAR2_2_trip AND AHU_FAR2_2_latch),Q=>AHU_FAR2_2_trip_error);
AHU_FAR2_2_common_alarm := AHU_FAR2_2_fire OR AHU_FAR2_2_gas OR AHU_FAR2_2_smoke OR AHU_FAR2_2_status_error OR AHU_FAR2_2_trip_error;


AHU_FAR2_common_alarm := AHU_FAR2_1_common_alarm OR AHU_FAR2_2_common_alarm ;
AHU_FAR2_dcs_occupied := AHU_FAR2_1_dcs_occupied OR AHU_FAR2_2_dcs_occupied;

	FB_AHU_FAR2(
	ON1:=AHU_FAR2_1_trigger ,
	ON2:=AHU_FAR2_2_trigger ,
	ON3:=FALSE ,
	status_error_1:= AHU_FAR2_1_status_error,
	status_error_2:=AHU_FAR2_2_status_error ,
	status_error_3:=FALSE ,
	trip_error_1:=AHU_FAR2_1_trip_error ,
	trip_error_2:=AHU_FAR2_2_trip_error ,
	trip_error_3:=FALSE ,
	Latch1:=AHU_FAR2_1_latch ,
	Latch2:=AHU_FAR2_2_latch ,
	Latch3:=AHU_FAR2_dummy ,
	DcsOccupied_1=>AHU_FAR2_1_dcs_occupied ,
	DcsOccupied_2=>AHU_FAR2_2_dcs_occupied ,
	DcsOccupied_3=> );


EF_FAR2_1A_status_Filter(IN:=(NOT EF_FAR2_1A_status AND EF_FAR2_1A_latch),Q=>EF_FAR2_1A_status_error);
EF_FAR2_1A_trip_Filter(IN:=(EF_FAR2_1A_trip AND EF_FAR2_1A_latch),Q=>EF_FAR2_1A_trip_error);
EF_FAR2_1A_common_alarm := EF_FAR2_1A_status_error OR EF_FAR2_1A_trip_error;



EF_FAR2_1B_status_Filter(IN:=(NOT EF_FAR2_1B_status AND EF_FAR2_1B_latch),Q=>EF_FAR2_1B_status_error);
EF_FAR2_1B_trip_Filter(IN:=(EF_FAR2_1B_trip AND EF_FAR2_1B_latch),Q=>EF_FAR2_1B_trip_error);
EF_FAR2_1B_common_alarm := EF_FAR2_1B_status_error OR EF_FAR2_1B_trip_error;


EF_FAR2_common_alarm := EF_FAR2_1A_common_alarm OR EF_FAR2_1B_common_alarm;
EF_FAR2_dcs_occupied := EF_FAR2_1A_dcs_occupied OR EF_FAR2_1B_dcs_occupied;

	FB_EF_FAR2(
	ON1:=EF_FAR2_1A_trigger ,
	ON2:=EF_FAR2_1B_trigger ,
	ON3:=FALSE ,
	status_error_1:= EF_FAR2_1A_status_error,
	status_error_2:=EF_FAR2_1B_status_error ,
	status_error_3:=FALSE ,
	trip_error_1:=EF_FAR2_1A_trip_error ,
	trip_error_2:=EF_FAR2_1B_trip_error ,
	trip_error_3:=FALSE ,
	Latch1:=EF_FAR2_1A_latch ,
	Latch2:=EF_FAR2_1B_latch ,
	Latch3:=EF_FAR2_dummy ,
	DcsOccupied_1=>EF_FAR2_1A_dcs_occupied ,
	DcsOccupied_2=>EF_FAR2_1B_dcs_occupied ,
	DcsOccupied_3=> );


(**************************)

EF_FAR2_3_status_Filter(IN:=(NOT EF_FAR2_3_status AND EF_FAR2_3_latch),Q=>EF_FAR2_3_status_error);
EF_FAR2_3_trip_Filter(IN:=(EF_FAR2_3_trip AND EF_FAR2_3_latch),Q=>EF_FAR2_3_trip_error);
EF_FAR2_3_common_alarm := EF_FAR2_3_status_error OR EF_FAR2_3_trip_error;


FB_EF_FAR2_3(
Trigger:=EF_FAR2_3_trigger ,
Latch:=EF_FAR2_3_latch ,
DCS_Occupied=>EF_FAR2_3_dcs_occupied );


(*************************)


EF_FAR2_2_status_Filter(IN:=(NOT EF_FAR2_2_status AND EF_FAR2_2_latch),Q=>EF_FAR2_2_status_error);
EF_FAR2_2_trip_Filter(IN:=(EF_FAR2_2_trip AND EF_FAR2_2_latch),Q=>EF_FAR2_2_trip_error);
EF_FAR2_2_common_alarm := EF_FAR2_2_status_error OR EF_FAR2_2_trip_error;


(***************************)

EDH_FAR2_1_on_status := AHU_FAR2_dcs_occupied;

FB_EDH_FAR2_1(on_status:= EDH_FAR2_1_on_status , flow_status:= EDH_FAR2_1_flow_status , high_temp:= EDH_FAR2_1_high_temp);

EDH_FAR2_1_hightemp_error := EDH_FAR2_1_high_temp;
EDH_FAR2_1_common_alarm := EDH_FAR2_1_hightemp_error;


(***************************)

common_alarm := AHU_FAR2_common_alarm OR EF_FAR2_common_alarm OR EF_FAR2_3_common_alarm OR EF_FAR2_2_common_alarm;

dcs_occupied := AHU_FAR2_dcs_occupied OR EF_FAR2_dcs_occupied OR EF_FAR2_3_dcs_occupied;
END_PROGRAM

(* POU NonProcessBuildingSubstation, ST *)
PROGRAM NonProcessBuildingSubstation
VAR
	AHU_NPBSS_common_alarm : BOOL;
	AHU_NPBSS_dcs_occupied : BOOL;

	AHU_NPBSS_dummy : BOOL;
	FB_AHU_NPBSS: Flowchart_3_4_CTRL;

	AHU_NPBSS_1_status AT%I* : BOOL;
	AHU_NPBSS_1_trip AT%I* : BOOL;
	AHU_NPBSS_1_mode AT%I* : BOOL;
	AHU_NPBSS_1_belt AT%I* : BOOL;
	AHU_NPBSS_1_fire AT%I* : BOOL;
	AHU_NPBSS_1_gas AT%I* : BOOL;
	AHU_NPBSS_1_smoke AT%I* : BOOL;

	AHU_NPBSS_1_trigger : BOOL;
	AHU_NPBSS_1_latch : BOOL;
	AHU_NPBSS_1_common_alarm : BOOL;
	AHU_NPBSS_1_status_error : BOOL;
	AHU_NPBSS_1_trip_error : BOOL;
	AHU_NPBSS_1_dcs_occupied : BOOL;

	AHU_NPBSS_1_status_Filter : ErrorFilter;
	AHU_NPBSS_1_trip_Filter : ErrorFilter;


	AHU_NPBSS_2_status AT%I* : BOOL;
	AHU_NPBSS_2_trip AT%I* : BOOL;
	AHU_NPBSS_2_mode AT%I* : BOOL;
	AHU_NPBSS_2_belt AT%I* : BOOL;
	AHU_NPBSS_2_fire AT%I* : BOOL;
	AHU_NPBSS_2_gas AT%I* : BOOL;
	AHU_NPBSS_2_smoke AT%I* : BOOL;

	AHU_NPBSS_2_trigger : BOOL;
	AHU_NPBSS_2_latch : BOOL;
	AHU_NPBSS_2_common_alarm : BOOL;
	AHU_NPBSS_2_status_error : BOOL;
	AHU_NPBSS_2_trip_error : BOOL;
	AHU_NPBSS_2_dcs_occupied : BOOL;

	AHU_NPBSS_2_status_Filter : ErrorFilter;
	AHU_NPBSS_2_trip_Filter : ErrorFilter;



(*****************************)


	EF_NPBSS_common_alarm : BOOL;
	EF_NPBSS_dcs_occupied : BOOL;

	EF_NPBSS_dummy : BOOL;
	FB_EF_NPBSS: Flowchart_3_4_CTRL;

	EF_NPBSS_1_status AT%I* : BOOL;
	EF_NPBSS_1_trip AT%I* : BOOL;
	EF_NPBSS_1_mode AT%I* : BOOL;

	EF_NPBSS_1_trigger : BOOL;
	EF_NPBSS_1_latch : BOOL;
	EF_NPBSS_1_common_alarm : BOOL;
	EF_NPBSS_1_status_error : BOOL;
	EF_NPBSS_1_trip_error : BOOL;
	EF_NPBSS_1_dcs_occupied : BOOL;

	EF_NPBSS_1_status_Filter : ErrorFilter;
	EF_NPBSS_1_trip_Filter : ErrorFilter;


	EF_NPBSS_2_status AT%I* : BOOL;
	EF_NPBSS_2_trip AT%I* : BOOL;
	EF_NPBSS_2_mode AT%I* : BOOL;

	EF_NPBSS_2_trigger : BOOL;
	EF_NPBSS_2_latch : BOOL;
	EF_NPBSS_2_common_alarm : BOOL;
	EF_NPBSS_2_status_error : BOOL;
	EF_NPBSS_2_trip_error : BOOL;
	EF_NPBSS_2_dcs_occupied : BOOL;

	EF_NPBSS_2_status_Filter : ErrorFilter;
	EF_NPBSS_2_trip_Filter : ErrorFilter;


(****************************************)


	EF_NPBSS_3_status AT%I* : BOOL;
	EF_NPBSS_3_trip AT%I* : BOOL;
	EF_NPBSS_3_mode AT%I* : BOOL;

	EF_NPBSS_3_trigger : BOOL;
	EF_NPBSS_3_latch : BOOL;
	EF_NPBSS_3_common_alarm : BOOL;
	EF_NPBSS_3_status_error : BOOL;
	EF_NPBSS_3_trip_error : BOOL;
	EF_NPBSS_3_dcs_occupied : BOOL;

	EF_NPBSS_3_status_Filter : ErrorFilter;
	EF_NPBSS_3_trip_Filter : ErrorFilter;

(*******************************************************)


	FB_EDH_NPBSS_3: Flowchart_5_6;
	EDH_NPBSS_3_on_status : BOOL;
	EDH_NPBSS_3_flow_status AT%I* : BOOL;
	EDH_NPBSS_3_high_temp AT%I* : BOOL;

	EDH_NPBSS_3_common_alarm : BOOL;
	EDH_NPBSS_3_hightemp_error : BOOL;


(*********************************************************)

	MD_NPBSS_1A_damper_open AT%I* : BOOL;
	MD_NPBSS_1A_damper_close AT%I* : BOOL;

	MD_NPBSS_1B_damper_open AT%I* : BOOL;
	MD_NPBSS_1B_damper_close AT%I* : BOOL;

	MD_NPBSS_1C_damper_open AT%I* : BOOL;
	MD_NPBSS_1C_damper_close AT%I* : BOOL;

	MD_EF_NPBSS_1D_damper_open AT%I* : BOOL;
	MD_EF_NPBSS_1D_damper_close AT%I* : BOOL;

(******************************************************)

	MFD_NPBSS_1_damper_open AT%I* : BOOL;
	MFD_NPBSS_1_damper_close AT%I* : BOOL;

	MFD_NPBSS_2_damper_open AT%I* : BOOL;
	MFD_NPBSS_2_damper_close AT%I* : BOOL;

	MFD_NPBSS_3_damper_open AT%I* : BOOL;
	MFD_NPBSS_3_damper_close AT%I* : BOOL;

	MFD_NPBSS_4_damper_open AT%I* : BOOL;
	MFD_NPBSS_4_damper_close AT%I* : BOOL;

	MFD_NPBSS_5_damper_open AT%I* : BOOL;
	MFD_NPBSS_5_damper_close AT%I* : BOOL;

